//external gridcode trip (Now coming from missing phase current/ high current unbalance).
IF set.e_InverterMode = eInvertermodes.Afe OR setMaster.b_ExtgridCodeTrip THEN
	ton_GridCodeTripDelay(IN := b_extGridCodetrip);
	setMaster.b_ExtgridCodeTrip := ton_GridCodeTripDelay.Q;
	setSlave.b_ExtgridCodeTrip := ton_GridCodeTripDelay.Q;
END_IF

//calculate internal loss offset
r_ActiveLossOffset := r_APloss;
r_ReactiveLossOffset:= r_RPloss + st_params.r_ReactiveOffset;


ton_RampDisabled(IN := get.b_StartedState);
//Gross power: requested + internal loss 
r_grossActivePower := set.r_ActivePower * st_params.r_ActiveSetpointGain - r_ActiveLossOffset;
fb_ramp_Pset(IN := r_grossActivePower, SETtoIN := ton_RampDisabled.Q);
//magic reactive fix to the inverter:P
//SEL(set.r_ReactivePower < 0, -0.00039, -0.0007) * -set.r_ReactivePower + 1;
r_grossReactivePower := st_params.r_ReactiveSetpointGain * set.r_ReactivePower - r_ReactiveLossOffset;
fb_ramp_Qset(IN := r_grossReactivePower, SETtoIN := ton_RampDisabled.Q, SetZero:= NOT get.b_StartedState);


//Powerlimiting mode ugrid
PowerLimitingMode(
	enable := get.b_InverterGridFormingMode AND NOT set.b_DisableShifting,
	PowerLimitingMode := set.e_PowerLimitingMode,
	ActivePower := get.r_ActivePower,
	MaxPower := set.r_Pmax,
	MinPower := set.r_Pmin,
	ShiftHoldTimeRemaining => get.t_ShiftHoldTimeRemaining,
	Active	=> get.Events.b_PlimitShiftingActive,
	Pmax => r_PmaxFinal,
	Pmin => r_PminFinal,
	FreqOffset => r_PLMfreqOffset,
	VoltOffset => r_PLMvoltOffset,
	st_params := st_params.FreqVoltageShift,
	);
	
//Max Charge Power
SetMaster.r_Pmin := r_PminFinal * r_PM1Load;
SetSlave.r_Pmin := r_PminFinal * r_PM2Load;
//Max Discharge Power
SetMaster.r_Pmax := r_PmaxFinal * r_PM1Load;
SetSlave.r_Pmax := r_PmaxFinal * r_PM2Load;
//Max AC current limit (first reactive limits, then active);
SetMaster.r_ACcurrentLimit := set.r_ACcurrentLimit * r_PM1Load;
SetSlave.r_ACcurrentLimit:= set.r_ACcurrentLimit * r_PM2Load;

//ActivePower
setMaster.r_ActivePower := SEL(set.r_Pmax = 0 AND fb_ramp_Pset.Q > 0, fb_ramp_Pset.Q * r_PM1Load, st_params.i_ChargeOnlyIdlePower); 
setSlave.r_ActivePower := fb_ramp_Pset.Q * r_PM2Load; 


//Set Reactive Power
setMaster.r_ReactivePower := fb_ramp_Qset.Q * r_PM1Load;// fb_ramp_Qset.Q  // fb_ramp_Qset.Q * r_PM1Load;
setSlave.r_ReactivePower := fb_ramp_Qset.Q * r_PM2Load; //fb_ramp_Qset.Q * r_PM2Load;

//Overcurrent factor
setMaster.r_overcurrentFactor := CoolingDerating();
setSlave.r_overcurrentFactor := CoolingDerating();

//Max power change rate
SetMaster.i_PowerChangeRate := st_params.i_MaxPowerChangeRate; //limit to 300%/s 
SetSlave.i_PowerChangeRate := st_params.i_MaxPowerChangeRate;

//set frequency to inverter
r_FreqDeltaLOM := FreqPulseDelta(LOM.b_enable AND settings.MachineParams.Powerstack.LOM.EnablePowerPulse,
								PulseSize := st_params.LOM.PowerPulseSize,
								Droop := get.r_FrequencyDroop, 
								DetectionTime := SEL(st_params.LOM.ForceSlowDetection, st_params.LOM.DetectionTimeFast_ms, st_params.LOM.DetectionTimeSlow_ms)
								);


		
								
setMaster.r_NomFrequency := set.r_NominalOutputFrequency + r_FreqDeltaLOM + r_PLMfreqOffset;
SetSlave.r_NomFrequency := set.r_NominalOutputFrequency + r_FreqDeltaLOM + r_PLMfreqOffset;


//set voltage to inverter
setMaster.r_NomVoltage := set.r_NominalOutputVoltage + r_PLMVoltOffset;
SetSlave.r_NomVoltage := set.r_NominalOutputVoltage + r_PLMvoltOffset;
END_METHOD

METHOD CoolingDerating : REAL

VAR_INST
	percentage			: REAL;
END_VAR
//Cooling derating
IF by_CoolingPowerRequest <> 2 AND get.b_ControlEnabled THEN
	percentage := LIMIT(0, 100 - st_params.ui_DeratingLimCooling, st_params.ui_OvercurrentRating);
	get.Events.b_CoolingDerating := TRUE;
ELSE
	percentage := st_params.ui_OvercurrentRating;
	get.Events.b_CoolingDerating := FALSE;
END_IF

CoolingDerating := percentage / 100;
END_METHOD

ACTION CoolingReady_active:
IF eControl <> stand_by THEN
	by_CoolingControl := 2;
END_IF

get.e_State := eStatusPowerStack.Wait_CoolingMode2;

SFCTIP := 	((by_CoolingPowerRequest > 1 AND NOT DetectConnectionLoss(TRUE)) OR 
			(eControl = stand_by AND by_CoolingPowerRequest =1)) AND NOT SFCTip;
END_ACTION

METHOD DetectConnectionLoss : BOOL
VAR_INPUT
	CurrentState		: BOOL;
END_VAR

VAR_INST
	ftrig_Input 	: F_TRIG;
	ftrig_Output 	: F_TRIG;
END_VAR
ftrig_Output(CLK := b_OutputConnected);
ftrig_Input(CLK:= b_InputConnected);

IF NOT b_OutputConnected AND ftrig_Input.Q THEN
	DetectConnectionLoss := TRUE;
END_IF


IF NOT b_InputConnected AND ftrig_Output.Q THEN
	DetectConnectionLoss := TRUE;
END_IF

IF CurrentState THEN
	DetectConnectionLoss := NOT (b_InputConnected OR b_OutputConnected);
END_IF
END_METHOD

METHOD PRIVATE DetectGridSync : BOOL
VAR_INPUT
	b_netconFB					: BOOL;
	b_InverterGridFormingMode	: BOOL;
	b_ExtGridConnected			: BOOL;
	b_ACOK						: BOOL;
	b_IsochroneMode				: BOOL;
	b_GridCodeActiveInverter 	: BOOL;
	b_GridCodeTripInverter		: BOOL;
	t_GridLostMaxTripTime		: TIME;
	t_GridOKReleaseTime			: TIME;
END_VAR

VAR_INST
	rTrigStartCommand			: R_TRIG;
	b_inverterGridCodeOK			: BOOL;
	b_AFErequested				: BOOL;
	ton_DetectionDelay			: TON := (PT := T#50MS);
	ton_DetectionDelayNoGrid	: TON := (PT := T#50MS);
	b_ExtGridCheck				: BOOL;
	tp_ExtGridLost				: TP := (PT := T#40MS);
	fTrig_ACOK					: F_TRIG;
	ton_GridLostRelease			: TON := (PT := T#0M);
	ton_GridTripDelay			: TON ;
	DisableGCtrip				: TOF := (PT:= T#1S);
END_VAR


VAR_IN_OUT
	b_Gridtied				: BOOL;
	b_GridCodeOK			: BOOL;
	b_gridCheckActive		: BOOL;
	b_ACdetected			: BOOL;
END_VAR
PowermoduleMaster.set.b_GridCodeEnable := st_params.b_GridCodesEnabled;

// update AC detected while not connected to busbar
b_ExtGridCheck := b_ExtGridConnected AND b_InverterGridFormingMode; // OLD: get.e_InverterMode = eInvertermodes.Afe;
ton_DetectionDelay(IN := NOT b_ACOK OR (b_netconFB AND NOT get.b_InverterRunning));
tp_ExtGridLost(IN := NOT b_ExtGridConnected, PT := TO_TIME(settings.GridParams.ui_GCTripMaxTripTime));
IF ton_DetectionDelay.Q OR NOT b_netconFB OR b_ExtGridCheck OR tp_ExtGridLost.Q THEN
	b_ACdetected	:= b_ACOK;
END_IF

//conditions where gridAC is not possible.
//ton_DetectionDelayNoGrid(IN := b_netconFB AND b_InverterGridFormingMode AND get.b_StartedState); // OLD: get.e_InverterMode = eInvertermodes.Afe;
//IF ton_DetectionDelayNoGrid.Q THEN
//	b_ACdetected := FALSE;
//END_IF

//Grid OK inverter statement
b_inverterGridCodeOK := NOT b_GridCodeActiveInverter OR (NOT b_GridCodeTripInverter AND b_GridCodeActiveInverter);

//disable GC Trip
DisableGCTrip(IN:= detectConnectionLoss(TRUE));


//Manual gridlost check
b_AFERequested := set.e_InverterMode = eInvertermodes.Afe;
b_gridCheckActive := b_AFERequested OR NOT b_gridCodeOK AND NOT DisableGCTrip.Q; //or not netconfb ;
//b_gridCheckActive := set.e_InverterMode = eInvertermodes.Afe AND get.b_ControlEnabled AND NOT DisableGCTrip.Q;

LOM(r_Freq := get.r_FrequencyD7, 
	r_NomFreq := set.r_NominalOutputFrequency, 
	r_Volt:= Get.r_ACVoltageD7,
	b_enable := Get.b_StartedState AND get.e_PowerMode = ePowermodes.Isochronous AND get.e_InverterMode <> eInvertermodes.Afe,
	SlowDetection:= set.b_slowLom, //only activate fast when external grid is coupled.
	st_params := st_params.LOM);

IF LOM.Q THEN
	b_gridCheckActive := TRUE;
END_IF

IF b_ACOK AND b_gridCodeOK THEN
	LOM.Reset();
END_IF


ton_GridTripDelay(IN:= NOT b_ACOK AND b_gridCheckActive, PT := t_GridLostMaxTripTime);
IF ton_GridTripDelay.Q OR NOT b_inverterGridCodeOK OR LOM.Q THEN
	b_ACdetected := FALSE;
	b_gridCodeOK := FALSE;
END_IF

get.t_GridCodeReconnectTime := ton_GridLostRelease.PT - ton_GridLostRelease.ET;

ton_GridLostRelease(
	IN := b_ACOK AND b_inverterGridCodeOK AND NOT LOM.Q AND NOT b_gridCodeOK,
	PT := SEL(b_gridCheckActive AND b_AFERequested, T#1S, t_GridOKReleaseTime)
	);

rTrigStartCommand(CLK:= eControl = start);
IF ton_GridLostRelease.Q OR NOT get.b_ControlEnabled OR DisableGCTrip.Q OR rTrigStartCommand.Q THEN
	b_gridCodeOK := TRUE;
END_IF

get.Events.b_GridCodeWarning := NOT b_gridCodeOK;
b_Gridtied := b_netconFB AND b_gridCodeOK AND b_gridCheckActive;
END_METHOD

METHOD PUBLIC EMstop : BOOL
EMstop := 
	SFCCurrentStep = 'Init' AND Netcontactor.Open() AND ShutdownFull(TRUE);
//Set internal control mode to shutdown
eControl := Shutdown;



//force SFC to init with execution of init step
SFCReset := TRUE;

IF EMstop THEN
	get.e_State := eStatusPowerStack.off;
END_IF
END_METHOD

METHOD FreqCheckPLimitUgrid : BOOL
VAR_INPUT
	b_enable			: BOOL;
	r_Frequency			: REAL;
	r_LowFreqLim		: REAL;
	r_HighFreqLim		: REAL;
	t_TriggerDelay		: TIME := T#1000MS;
END_VAR

VAR_OUTPUT
	b_LowFreqTrip		: BOOL;
	b_HighFreqTrip		: BOOL;
END_VAR

VAR_INST
	ton_TriggerDelay	: TON;
	Activate			: BOOL;
END_VAR
(*
-------INFO---------
This function is added to raise a normal shutdown before the inverter does at under/over frequency in ugrid.
this under/over frequency check is raised when the pmax or pmin limit is reached in ugrid mode resulting in frequency shift done by inverter.
To avoid a trip by inverter underfrequency, resulting in ac outage, we detect the event slightly earlier.
This creates a normal shutdown command in the error program and will keep possibility of correctly stopping the cooling supply.
If this script was not here, the under frequency trip of the inverter would be seen, leading to AC outage and this
interrupts all internal AC devices. Especially for the heatpump, this is undesirable. 
*)


activate := b_enable AND LIMIT(get.r_Pmin, get.r_ActivePower, get.r_Pmax) <> get.r_ActivePower; 
ton_triggerDelay(IN := (r_Frequency < r_LowFreqLim OR r_Frequency > r_HighFreqLim) AND activate, PT := t_TriggerDelay);

IF ton_triggerDelay.Q THEN
	b_LowFreqTrip := r_Frequency < r_LowFreqLim;
	b_HighFreqTrip := r_Frequency > r_HighFreqLim;
END_IF
END_METHOD

METHOD FreqPulseDelta : REAL
VAR_INPUT
	Enable			: BOOL;
	PulseSize		: REAL; // % of ratedpower
	Droop			: REAL;
	DetectionTime	: UINT;
END_VAR

VAR_INST
	DetectionTimeFactor	: UINT := 3; 
	FreqShift			: REAL;
	ton_PulseTime		: TON;
	b_toggleState		: BOOL;
END_VAR
(*-------INFO---------
This function is for intentionally disturbing the frequency setpoint of the inverter in a microgrid. It has been with grid and genset connected.
Testing must be done for multiple batteries in ugrid mode. The small disturbances are made on the frequency. The pulsesize is in % of rated power.
The change of the frequency therefore is relative to the droop settings and the nominal frequency setting.
The detection time and a multiplication factor gives the sweet spot of the pulse time and detection mechanism in the LOM detection.

If this puls is disabled in ugrid, the LOM detection might not function properly and
frequency might drift away in case of grid loss before transition to island mode is made.
*)

ton_PulseTime(IN := NOT ton_pulseTime.Q, PT := TO_TIME(detectionTime*DetectionTimeFactor)); //must be bigger than detection time. factor 5 seems fine.

IF ton_pulseTime.Q THEN
	b_ToggleState := NOT b_toggleState;
END_IF


FreqShift := PulseSize / 100 * settings.GridParams.r_GridNominalFrequency * Droop / 100; 
IF enable THEN
	FreqPulseDelta := SEL(b_toggleState, -1, 1) * FreqShift;
ELSE
	FreqPulseDelta := 0;
END_IF
END_METHOD

METHOD PUBLIC GetDiagnostics
VAR_IN_OUT
	AddError		: ARRAY [*] OF FB_AddErrorST;
	a_ActiveEvents	: ARRAY [*] OF ST_ErrorStruct;
	w_Index			: WORD;
END_VAR

VAR_INST
	varString		: STRING;
END_VAR
(*POWERSTACK*)
	//Warnings
	(*DC voltage diff*) 	AddError[w_Index](
			b_ErrorTrig			:= Get.Events.b_DCdeviationHigh,
			out_ST_Error			:= a_ActiveEvents[w_Index],
			w_ErrorID					:= 1,
			e_ObjectID				:= eObject_ID.PowerStack,
			s_Message				:= 'DC voltage difference between powermodules high',
			e_sev					:= eseverity.Warning
			);
		w_Index := w_Index +1;
	
	(*Temperature*) 			AddError[w_Index](
			b_ErrorTrig			:= Get.Events.b_TemperatureDeviationHigh,
			out_ST_Error			:= a_ActiveEvents[w_Index],
			w_ErrorID					:= 2,
			e_ObjectID				:= eObject_ID.PowerStack,
			s_Message				:= 'temperature difference between powermodules high',
			e_sev					:= eseverity.Warning,
			b_AutoClear			:= TRUE,
		);
		w_Index := w_Index +1;
		
	(*UnderFreq limit exceeded*)	AddError[w_Index](
			b_ErrorTrig				:= Get.Events.b_UnderFreqFault ,
			out_ST_Error			:= a_ActiveEvents[w_Index],
			w_ErrorID				:= 3,
			e_ObjectID				:= eObject_ID.PowerStack,
			s_Message				:= 'under frequency trip',
			e_sev					:= eseverity.normalshutdown
		);
		w_Index := w_Index +1;	
		
	(*OverFreq limit exceeded*)		AddError[w_Index](
			b_ErrorTrig				:= Get.Events.b_OverFreqFault,
			out_ST_Error			:= a_ActiveEvents[w_Index],
			w_ErrorID				:= 4,
			e_ObjectID				:= eObject_ID.PowerStack,
			s_Message				:= 'over frequency trip',
			e_sev					:= eseverity.normalshutdown
		);
		w_Index := w_Index +1;	
		
	(*Cooling derating*)	AddError[w_Index](
			b_ErrorTrig			:=  get.Events.b_CoolingDerating,
			out_ST_Error			:= a_ActiveEvents[w_Index],
			w_ErrorID				:= 5,
			s_Message				:= 'Cooling system derating causing inverter output to be limited',
			e_sev					:= eseverity.warning,
			b_autoclear				:= TRUE,
		);
		w_Index := w_Index +1;

	(*SFC Timeout*)	AddError[w_Index](
			b_ErrorTrig				:= SFCerror,
			out_ST_Error			:= a_ActiveEvents[w_Index],
			w_ErrorID				:= 6,
			e_ObjectID				:= eObject_ID.PowerStack,
			s_Message				:= CONCAT('SFC error at step: ', s_errorstep),
			e_sev					:= eseverity.NormalShutdown
		);
		w_Index := w_Index +1;
		
		
(*Start inhibit*)	AddError[w_Index](
			b_ErrorTrig				:= NOT get.b_StartEnabled AND set.e_InverterMode = eInvertermodes.Afe,
			out_ST_Error			:= a_ActiveEvents[w_Index],
			w_ErrorID				:= 8,
			s_Message				:= CONCAT('Inverter starting in grid following mode inhibited, ',SEL(NOT get.b_GridCodeOK AND get.b_GridCodeCheckActive, 'waiting for grid AC','waiting for gridcode release')),
			e_sev					:= eseverity.info,
			b_autoclear				:= TRUE,
		);
		w_Index := w_Index +1;
		
(*Start inhibit*)	AddError[w_Index](
			b_ErrorTrig			:= NOT get.b_StartEnabled AND set.e_InverterMode = eInvertermodes.Island,
			out_ST_Error			:= a_ActiveEvents[w_Index],
			w_ErrorID				:= 9,
			s_Message				:= 'Inverter starting in grid forming mode inhibited, disconnect AC from busbar',
			e_sev					:= eseverity.info,
			b_autoclear				:= TRUE,
		);
		w_Index := w_Index +1;
		
	(*Overvoltage fault*)	AddError[w_Index](
			b_ErrorTrig			:= get.Events.b_OverVoltageFault,
			out_ST_Error			:= a_ActiveEvents[w_Index],
			w_ErrorID				:= 10,
			s_Message				:= 'Overvoltage fault', //10-12-2024: change to normalshutdown once verified
			e_sev					:= eseverity.warning,
			b_autoclear				:= FALSE,
		);
		w_Index := w_Index +1;
		
	(*underVoltage fault*)	AddError[w_Index](
			b_ErrorTrig			:= get.Events.b_underVoltageFault,
			out_ST_Error			:= a_ActiveEvents[w_Index],
			w_ErrorID				:= 11,
			s_Message				:= 'Undervoltage fault',
			e_sev					:= eseverity.warning, // 10-12-2024: change to normalshutdown once verified 
			b_autoclear				:= FALSE,
		);
		w_Index := w_Index +1;
		
	(*Overvoltage warning*)	AddError[w_Index](
			b_ErrorTrig			:= get.Events.b_OverVoltageFault,
			out_ST_Error			:= a_ActiveEvents[w_Index],
			w_ErrorID				:= 12,
			s_Message				:= 'Overvoltage warning',
			e_sev					:= eseverity.warning,
			b_autoclear				:= TRUE,
		);
		w_Index := w_Index +1;
		
	(*underVoltage fault*)	AddError[w_Index](
			b_ErrorTrig			:= get.Events.b_underVoltageFault,
			out_ST_Error			:= a_ActiveEvents[w_Index],
			w_ErrorID				:= 13,
			s_Message				:= 'Undervoltage warning',
			e_sev					:= eseverity.warning,
			b_autoclear				:= TRUE,
		);
		w_Index := w_Index +1;

		(*Overvoltage warning*)	AddError[w_Index](
			b_ErrorTrig			:= get.Events.b_TemperatureFault,
			out_ST_Error			:= a_ActiveEvents[w_Index],
			w_ErrorID				:= 14,
			s_Message				:= 'Temperature fault',
			e_sev					:= eseverity.warning,
			b_autoclear				:= TRUE,
		);
		w_Index := w_Index +1;
		
	(*underVoltage fault*)	AddError[w_Index](
			b_ErrorTrig			:= get.Events.b_TemperatureWarning,
			out_ST_Error			:= a_ActiveEvents[w_Index],
			w_ErrorID				:= 15,
			s_Message				:= 'Temperature warning',
			e_sev					:= eseverity.warning,
			b_autoclear				:= TRUE,
		);
		w_Index := w_Index +1;
		
(*Plimit warning*)	AddError[w_Index](
			b_ErrorTrig				:= get.Events.b_PlimitShutdownWarning,
			out_ST_Error			:= a_ActiveEvents[w_Index],
			w_ErrorID				:= 16,
			s_Message				:= CONCAT(CONCAT('Power limit reached, shutdown in ', TO_STRING(get.Events.ui_shutdownRemainingTime)),'s'),
			e_sev					:= eseverity.warning,
			b_autoclear				:= TRUE,
		);
		w_Index := w_Index +1;
		
(*Plimit shutdown*)	AddError[w_Index](
			b_ErrorTrig				:= get.Events.b_PlimitShutdown,
			out_ST_Error			:= a_ActiveEvents[w_Index],
			w_ErrorID				:= 17,
			s_Message				:= 'Power limit shutdown',
			e_sev					:= eseverity.normalshutdown,
			b_autoclear				:= TRUE,
		);
		w_Index := w_Index +1;
		
(*Plimit shifting *)	AddError[w_Index](
			b_ErrorTrig				:= get.Events.b_PlimitShiftingActive,
			out_ST_Error			:= a_ActiveEvents[w_Index],
			w_ErrorID				:= 18,
			s_Message				:= CONCAT(CONCAT(TO_STRING(set.e_PowerLimitingMode), ' active, output on hold for: '), TO_STRING(get.t_ShiftHoldTimeRemaining)),
			e_sev					:= eseverity.Warning,
			b_autoclear				:= TRUE,
		);
		w_Index := w_Index +1;

		
IF get.b_GridACdetected THEN
	varstring := CONCAT('gridcode disconnect active, reconnecting in: ', TO_STRING(get.t_GridCodeReconnectTime));
ELSE
	varstring := 'gridcode disconnect active, reset to reconnect in island mode';
END_IF
		
(*Gridcode disconnect *)	AddError[w_Index](
			b_ErrorTrig				:= get.Events.b_GridCodeWarning,
			out_ST_Error			:= a_ActiveEvents[w_Index],
			w_ErrorID				:= 19,
			s_Message				:= varstring,
			e_sev					:= eseverity.warning,
			b_autoclear				:= TRUE,
		);
		w_Index := w_Index +1;



(*INSERT NESTED OBJECTS*)
Netcontactor.GetDiagnostics(AddError := AddError, a_activeEvents:= a_ActiveEvents, w_Index:= w_Index);
PowermoduleMaster.GetDiagnostics(AddError := AddError, a_activeEvents:= a_ActiveEvents, w_Index:= w_Index);
PowermoduleSlave.GetDiagnostics(AddError := AddError, a_activeEvents:= a_ActiveEvents, w_Index:= w_Index);
END_METHOD

METHOD GetWearCounters : BOOL
VAR_INST
	RightNetContactor	:	FB_Varlogger;
	LeftNetContactor	:	FB_Varlogger;
	
	MasterPmMCCB		:	FB_Varlogger;
	MasterPmDCMain		:	FB_Varlogger;
	MasterPmPrecharge	:	FB_Varlogger;
	MasterPMACFanHrs	:	FB_Varlogger;		
	
	SlavePmMCCB			:	FB_Varlogger;
	SlavePmDCMain		:	FB_Varlogger;
	SlavePmPrecharge	:	FB_Varlogger;
	SlavePMACFan		:	FB_Varlogger;
	
	SlowDataTimer				:	TON := (PT := T#30M);
	
	initdone		:	Bool;
END_VAR
SlowDataTimer(in := NOT SlowDataTimer.Q);

IF get.PowermoduleMaster.w_OperationHours > 0 THEN
	Wearlogging.SetInteger(eLogItemGroupID.PowerStack, 	'MstrInvHrs', 				eLogTypes.WriteValue, 		WORD_TO_LINT(get.PowermoduleMaster.w_OperationHours));
END_IF
Wearlogging.SetFloat(eLogItemGroupID.PowerStack, 	'MstrMaxDischCurrentEver', 	eLogTypes.KeepHighestValue, REAL_TO_LREAL(get.PowermoduleMaster.r_ACCurrent));
Wearlogging.SetFloat(eLogItemGroupID.PowerStack, 	'MstrMaxChargeCurrentEver', eLogTypes.KeepLowestValue, 	REAL_TO_LREAL(get.PowermoduleMaster.r_AcCurrent));
		
												
MasterPmMCCB(			TriggerInput := get.PowermoduleMaster.b_MccbFb, 
						LogItemGroup :=  eLogItemGroupID.PowerStack, 
						LogItemName := 'MstrMCCBCnt', 
						LogType := eLogTypes.TrackCycles);	
						
MasterPmDCMain(			TriggerInput := get.PowermoduleMaster.b_DCcontactorFb, 
						LogItemGroup :=  eLogItemGroupID.PowerStack, 
						LogItemName := 'MstrDcMainCnt', 
						LogType := eLogTypes.TrackCycles);							

MasterPmPrecharge(		TriggerInput := get.PowermoduleMaster.b_PrechargeContactor, 
						LogItemGroup :=  eLogItemGroupID.PowerStack, 
						LogItemName := 'MstrDcPrechargeCnt', 
						LogType := eLogTypes.TrackCycles);		

MasterPMACFanHrs(		TriggerInput := get.PowermoduleMaster.b_FanFb, 
						LogItemGroup :=  eLogItemGroupID.PowerStack, 
						LogItemName := 'MstrAcFanHrs', 
						LogType := eLogtypes.TrackOnTime);	



					
IF b_doublePowermodule THEN
	Wearlogging.SetInteger(eLogItemGroupID.PowerStack, 	'SlvInvHrs', 				eLogTypes.WriteValue, 		WORD_TO_LINT(get.PowermoduleSlave.w_OperationHours));
	Wearlogging.SetFloat(eLogItemGroupID.PowerStack, 	'SlvMaxDischCurrentEver', 	eLogTypes.KeepHighestValue, REAL_TO_LREAL(get.PowermoduleSlave.r_ACCurrent));
	Wearlogging.SetFloat(eLogItemGroupID.PowerStack, 	'SlvMaxChargeCurrentEver', 	eLogTypes.KeepLowestValue, 	REAL_TO_LREAL(get.PowermoduleSlave.r_AcCurrent));		
												
	SlavePmMCCB(			TriggerInput := get.PowermoduleSlave.b_MccbFb, 
							LogItemGroup :=  eLogItemGroupID.PowerStack, 
							LogItemName := 'SlvMCCBCnt', 
							LogType := eLogTypes.TrackCycles);	
							
	SlavePmDCMain(			TriggerInput := get.PowermoduleSlave.b_DCcontactorFb, 
							LogItemGroup :=  eLogItemGroupID.PowerStack, 
							LogItemName := 'SlvDcMainCnt', 
							LogType := eLogTypes.TrackCycles);							
	
	SlavePmPrecharge(		TriggerInput := get.PowermoduleSlave.b_PrechargeContactor, 
							LogItemGroup :=  eLogItemGroupID.PowerStack, 
							LogItemName := 'SlvDcPrechargeCnt', 
							LogType := eLogTypes.TrackCycles);		
	
	SlavePMACFan(			TriggerInput := get.PowermoduleSlave.b_FanFb, 
							LogItemGroup :=  eLogItemGroupID.PowerStack, 
							LogItemName := 'SlvAcFanHrs', 
							LogType := eLogTypes.TrackOnTime);	
END_IF


RightNetContactor(		TriggerInput := get.Netcontactor.b_NetcontRightFb, 
						LogItemGroup :=  eLogItemGroupID.PowerStack, 
						LogItemName := 'NetcRightCnt', 
						LogType := eLogTypes.TrackCycles);		
												
LeftNetContactor(		TriggerInput := get.Netcontactor.b_NetcontLeftFb, 
						LogItemGroup :=  eLogItemGroupID.PowerStack, 
						LogItemName := 'NetcLeft', 
						LogType := eLogTypes.TrackCycles);	
						
IF NOT initdone THEN
	Wearlogging.SetFloat(eLogItemGroupID.General, 	'nameplatePowerCapacity', 	eLogTypes.WriteValue, 	TO_DINT(SEL(settings.Configuration.b_DoublePowerModule, 360, 720)));
	initdone := TRUE;		
END_IF
END_METHOD

METHOD PRIVATE InternalAcCheck : BOOL
VAR_INPUT
	r_ACVoltage	: REAL;
	r_ACFreq	: REAL;
END_VAR

VAR_INST
	b_VoltageOK				: BOOL;
	b_FrequencyOK			: BOOL;
	tof_ReleaseACNOK		: TOF := (PT:= T#2S);
	
	tof_MaxRetryTimeOut		: Tof := (PT:= T#60S);
	ton_ResetRetries		: TON := (PT:= T#60S);
	by_maxRetries			: BYTE := 5;
	by_retries				: BYTE;
	r_trigOK				: r_TRIG;
END_VAR
b_VoltageOK	:= LIMIT(350, r_ACVoltage, 450) = r_ACVoltage;
b_FrequencyOK :=  LIMIT(45, r_ACFreq, 65) = r_ACFreq;

tof_ReleaseACNOK(IN:= b_VoltageOK AND b_FrequencyOK); 
	
r_trigOK(CLK := tof_ReleaseACNOK.Q);
IF r_trigOK.Q THEN
	by_Retries := by_retries + 1;
END_IF
IF by_Retries > by_MaxRetries THEN
	by_Retries := 0;
	tof_MaxRetryTimeOut(IN := TRUE);
ELSE
	tof_MaxRetryTimeOut(IN := FALSE);
END_IF
	
InternalAcCheck := tof_ReleaseACNOK.Q AND NOT tof_MaxRetryTimeOut.Q;
ton_ResetRetries(IN:= InternalAcCheck);
IF ton_ResetRetries.Q THEN
	by_Retries := 0;
END_IF
END_METHOD

METHOD PowerLimitingMode;
VAR_INPUT
	enable					: BOOL;
	PowerLimitingMode		: ePLM;
	ActivePower				: REAL;
	MaxPower				: REAL;
	MinPower				: REAL;
END_VAR
VAR_IN_OUT CONSTANT
	st_params : ST_powerstack_ShiftingParams;
END_VAR

VAR_INST
	tof_shiftHoldTime	: Tof := (PT := T#20M);
	tPulseRate			: TIME := T#100MS;
	tonIncreasePulse	: TON := (PT := T#100MS);
	OffsetCounter		: CTUD;
	i_counterValue		: INT;
	PDeadband			: REAL := 3;
	PmaxReached			: BOOL;
	PminReached			: BOOL;
	Nolimit				: BOOL;
	
	MaxVoltOffsetUp		: REAL := 40;
	MaxVoltOffsetDown	: REAL := 40;
	
	MaxFreqOffsetUp		: REAL := 2.5;
	MaxFreqOffsetDown	: REAL := 2.5;
	
	r_FreqStepUp	: REAL := 0.1; // hz/s
	r_FreqStepDown	: REAL := 0.1; // hz/s
	r_FreqStepActual: REAL ;
	r_VoltStepUp	: REAL := 0.1; // V/s
	r_VoltStepDown 	: REAL := 0.1;
	r_VoltStepActual: REAL ;
	
	w_CounterSteps		: WORD := 1000;
	ton_InitialPmaxDelay	: TON := (PT := T#1S);
	ton_InitialPminDelay	: TON := (PT := T#1S);
	ton_shutdownTimer	: TON := (PT := T#1M);
	shutdownTrigger		: BOOL;
END_VAR

VAR_OUTPUT
	ShiftHoldTimeRemaining 	: TIME;
	Active				: BOOL;
	Pmax				: REAL;
	Pmin				: REAL;
	FreqOffset			: REAL;
	VoltOffset			: REAL;
END_VAR
IF NOT enable THEN
	Pmax := MaxPower;
	Pmin := MinPower;
	get.Events.b_PlimitShutdownWarning := FALSE;
	get.Events.b_PlimitShutdown := FALSE;
	active := FALSE;
	ShiftHoldTimeRemaining := st_params.ShiftingHoldTime;
	RETURN;
END_IF

shutdownTrigger	:= FALSE;
ton_InitialPmaxDelay(in := ActivePower > MAX(MaxPower, PDeadband), pt := st_params.InitialOverloadDelay);
ton_InitialPminDelay(in := ActivePower < MIN(MinPower, -PDeadband), pt := st_params.InitialOverloadDelay);

PmaxReached := ton_InitialPmaxDelay.Q;
PminReached	:= ton_InitialPminDelay.Q;

Nolimit := NOT PmaxReached AND NOT PminReached;

//max voltage offsets based on grid settings
MaxVoltOffsetUp := LIMIT(settings.GridParams.r_GridNominalVoltage, st_params.VoltMaxPu * settings.GridParams.r_GridNominalVoltage, settings.GridParams.r_GridvoltageMax) - settings.GridParams.r_GridNominalVoltage;
MaxVoltOffsetDown := settings.GridParams.r_GridNominalVoltage - LIMIT(settings.GridParams.r_GridvoltageMin, st_params.VoltMinPu * settings.GridParams.r_GridNominalVoltage, settings.GridParams.r_GridNominalVoltage);
r_VoltStepUp := MaxVoltOffsetUp / MAX(1, w_CounterSteps);
r_VoltStepDown := MaxVoltOffsetDown/ MAX(1, w_CounterSteps);
r_VoltStepActual := SEL(i_countervalue < 0, r_VoltStepUp, r_VoltStepDown);

//max frequency offsets based on grid settings
MaxFreqOffsetUp := LIMIT(settings.GridParams.r_GridNominalFrequency, st_params.FreqMaxPu * settings.GridParams.r_GridNominalFrequency, settings.GridParams.r_GridFrequencyMax) - settings.GridParams.r_GridNominalFrequency;
MaxFreqOffsetDown := settings.GridParams.r_GridNominalFrequency - LIMIT(settings.GridParams.r_GridFrequencyMin, st_params.FreqMinPu * settings.GridParams.r_GridNominalFrequency, settings.GridParams.r_GridNominalFrequency);
r_FreqStepUp := MaxFreqOffsetUp / MAX(1, w_CounterSteps);
r_FreqStepDown := MaxFreqOffsetDown / MAX(1, w_CounterSteps);
r_FreqStepActual := SEL(i_countervalue < 0, r_FreqStepUp, r_FreqStepDown);

//If shifting is done and limit is released. Hold current counter for 20 min, before reducing.
tof_shiftHoldTime(IN := (i_countervalue <> 0 AND NOT Nolimit), PT := st_params.ShiftingHoldTime);

//pulse Timer
tonIncreasePulse(IN := NOT tonIncreasePulse.Q, PT := tPulseRate);

OffsetCounter(
	CU := ((PminReached OR (i_countervalue < 0 AND Nolimit AND NOT tof_shiftHoldTime.Q)) AND tonIncreasePulse.Q) AND NOT OffsetCounter.QU,
	CD := ((PmaxReached OR (i_countervalue > 0 AND Nolimit AND NOT tof_shiftHoldTime.Q)) AND tonIncreasePulse.Q) AND NOT OffsetCounter.QD,
	LOAD := NOT get.b_StartedState,
	PV := SEL(get.b_StartedState, w_CounterSteps, w_CounterSteps*2));
i_countervalue := OffsetCounter.CV - w_CounterSteps;

CASE PowerLimitingMode OF
	ePLM.FreqShift: //default controlled by inverters
		Pmax := get.r_RatedPower;
		Pmin := -get.r_RatedPower;
		FreqOffset := LIMIT(-MaxFreqOffsetDown, r_FreqStepActual * i_countervalue, MaxFreqOffsetUp);
		
	ePLM.VoltShift:
		VoltOffset := LIMIT(-MaxVoltOffsetDown, r_VoltStepActual * i_countervalue, MaxVoltOffsetUp);
		Pmax := get.r_RatedPower;
		Pmin := -get.r_RatedPower;
		
	ePLM.FreqVoltShift:
		VoltOffset := LIMIT(-MaxVoltOffsetDown, r_VoltStepActual * i_countervalue, MaxVoltOffsetUp);
		FreqOffset := LIMIT(-MaxFreqOffsetDown, r_FreqStepActual * i_countervalue, MaxFreqOffsetUp);
		Pmax := get.r_RatedPower;
		Pmin := -get.r_RatedPower;
		
	ePLM.Shutdown:
		shutdownTrigger	:= NOT Nolimit;
		Pmax := get.r_RatedPower;
		Pmin := -get.r_RatedPower;	
END_CASE

ton_shutdownTimer(IN:= shutdownTrigger AND get.b_StartedState, PT := st_params.ShutdownDelay);
IF get.Events.b_PlimitShutdownWarning THEN
	get.Events.ui_shutdownRemainingTime := TO_UINT(TO_REAL(ton_shutdownTimer.PT - ton_shutdownTimer.ET)/ 1000);
END_IF

//outputs and events
Active := i_countervalue <> 0 AND PowerLimitingMode <> ePLM.Shutdown;
ShiftHoldTimeRemaining := tof_shiftHoldTime.PT - tof_shiftHoldTime.ET;
get.Events.b_PlimitShutdownWarning := ton_shutdownTimer.IN;
get.Events.b_PlimitShutdown := ton_shutdownTimer.Q;
END_METHOD

METHOD PUBLIC Reset : BOOL
Reset := Netcontactor.Reset() AND PowermoduleMaster.Reset() AND PowerModuleSlave.Reset() AND get.e_State <> eStatusPowerstack.fault;

standbyDeactivateState := FALSE;
get.b_GridCodeOK := TRUE;
//rs_Stop.RESET1 := TRUE;
//rs_StartUp.RESET1:= TRUE;	
//rs_Shutdown.RESET1:= TRUE;
END_METHOD

METHOD PRIVATE SetEvents
VAR_IN_OUT
	events							: ST_PowerStack_Events;
END_VAR

VAR_IN_OUT CONSTANT
	st_params						: ST_Powerstack_Params;
END_VAR


VAR
	r_DCVoltageDeviation			: REAL := 0.02; //2%
	r_TemperatureDeviation			: REAL:= 10; // 10C
END_VAR

VAR_INST
	tp_ACdetectionCheck				: TON:= (PT:=T#2S);
END_VAR
IF b_doublePowermodule THEN
	//DC Voltage Deviation higher than 2% between powermodules
	events.b_DCdeviationHigh:= ABS(get.PowermoduleMaster.r_DCVoltage - get.PowermoduleSlave.r_DCVoltage) > get.r_DCVoltage * r_DcVoltageDeviation;
	
	//Temperature Deviation between highest temperature in powermodules higher than 10C
	events.b_temperatureDeviationHigh:= ABS(get.PowermoduleMaster.r_TemperatureMax - get.PowermoduleSlave.r_TemperatureMax) > r_TemperatureDeviation;
	
	//slave warning and faults
	events.b_SlaveFault := get.PowermoduleSlave.Events.b_GeneralFaultFlag;
	events.b_SlaveWarning := get.PowermoduleSlave.Events.b_GeneralWarningFlag;

END_IF

//Master warning and faults
events.b_MasterFault := get.PowermoduleMaster.Events.b_GeneralFaultFlag;
events.b_MasterWarning := get.PowermoduleMaster.Events.b_GeneralWarningFlag;
events.b_OvercurrentFault := get.PowermoduleMaster.Events.b_F1OverCurrent OR get.PowermoduleSlave.Events.b_F1OverCurrent;
events.b_OvercurrentWarning := get.r_LoadPercent > get.r_OvercurrentValueAct * 100;
events.b_OvervoltageFault :=  get.PowermoduleMaster.Events.b_F2OverVoltage OR get.PowermoduleSlave.Events.b_F2OverVoltage;
events.b_OvervoltageWarning := get.r_ACVoltageD7 > settings.GridParams.r_GridvoltageMax;
events.b_TemperatureFault := PowermoduleMaster.GetTemperatureEvents(FALSE) OR
	PowermoduleSlave.GetTemperatureEvents(FALSE);
events.b_TemperatureWarning := PowermoduleMaster.GetTemperatureEvents(TRUE) OR
	PowermoduleSlave.GetTemperatureEvents(TRUE);
events.b_startupTimeOut := SFCerror;

FreqCheckPLimitUgrid(
	b_enable := get.b_StartedState AND get.e_InverterMode <> eInvertermodes.Afe AND get.e_PowerMode <> ePowermodes.Isochronous, 
	r_Frequency := get.r_FrequencySupply,
	r_LowFreqLim := st_params.r_FreqLowLimit,
	r_HighFreqLim := st_params.r_FreqHighLimit,
	t_TriggerDelay := TO_TIME(st_params.ui_FreqLimitTripDelay),
	b_LowFreqTrip => events.b_UnderFreqFault,
	b_HighFreqTrip => events.b_OverFreqFault);
END_METHOD

METHOD Shutdowncmd : BOOL
eControl := Shutdown;
//if SFC transition occurs, give feedback.
SFCreset := TRUE;
Shutdowncmd := FALSE;

get.e_State := eStatusPowerStack.shutdown; 
by_CoolingControl := 0;

IF b_InternalACRequired THEN
	get.e_State := eStatusPowerStack.Cooling_Shutdown;
	standbyDeactivateState := TRUE;
		powermodulemaster.Run(Powermode := ePowermodes.Isochronous, InverterMode := eInvertermodes.Microgrid, TRUE );
		IF netcontactor.Open() THEN;
			powermodulemaster.Run(Powermode := ePowermodes.DroopZeroStart, InverterMode := eInvertermodes.Microgrid, TRUE);
			Shutdowncmd	:= TRUE;
		END_IF
	//END_IF
ELSE
	IF ShutdownFull(FALSE)  THEN;
		IF Netcontactor.Open() THEN
			Shutdowncmd	:= TRUE;
			get.e_State := eStatusPowerStack.off;
		END_IF
	END_IF
	
END_IF
	
//	CASE by_CoolingPowerRequest OF // when cooling system allows, all power is killed
//		0: //off
//			by_CoolingControl := 0;
//				IF ShutdownFull(FALSE)  THEN ;
//					IF NOT st_params.b_StandbyEnable THEN
//						IF Netcontactor.Open() THEN
//							Shutdowncmd	:= TRUE;
//							get.e_State := eStatusPowerStack.off;
//						END_IF
//					ELSE			
//						IF NOT get.b_ACDetected THEN
//							Netcontactor.Open();
//						END_IF
//						Shutdowncmd	:= TRUE;
//						get.e_State := eStatusPowerStack.off;
//					END_IF
//				END_IF	
		
//		1, 2: //limited 	
////			IF false then //get.b_GridACdetected THEN //get.b_ACDetected THEN 
////				by_CoolingControl := 0;
////				Shutdowncmd := ShutdownFull(FALSE);
////			ELSE
//				by_CoolingControl := 1;
//				PowerModuleSlave.Shutdown(b_force := FALSE);
//				Shutdowncmd := Netcontactor.Open();
//			//END_IF// if cooling system still wants power AND AC grid is available	
//	END_CASE				

//Shutdowncmd := get.e_Status = eStatusPowerStack.off OR get.e_Status = eStatusPowerStack.init;
END_METHOD

METHOD PRIVATE ShutdownFull : BOOL
VAR_INPUT
	b_force : BOOL;
END_VAR

VAR_INST
	shutdownfb: BOOL;
	ton_ShutdownTimeOut				: TON:= (PT:=T#30S);
END_VAR
shutdownfb := PowermoduleMaster.Shutdown(b_force) AND PowermoduleSlave.Shutdown(b_force);
IF shutdownfb THEN
	st_InternalPsuSupplyRequest.b_Demand_HVDC := FALSE;
	st_InternalPsuSupplyRequest.b_Demand_24V := FALSE;
END_IF

ton_ShutdownTimeOut(IN := NOT shutdownfb, Q => get.Events.b_ShutdownTimeOut);


ShutdownFull := shutdownfb;
END_METHOD

METHOD Standbycmd : BOOL
VAR_INPUT
END_VAR
IF NOT(get.e_State = eStatusPowerstack.fault) THEN
	eControl := stand_by;
END_IF

//if SFC transition occurs, give feedback.
Standbycmd := get.e_State = eStatusPowerstack.Standby_GridSupply OR get.e_State = eStatusPowerstack.Standby_GridSupply;
END_METHOD

METHOD PUBLIC Startcmd : BOOL
IF get.b_StartEnabled THEN
	eControl := start;
END_IF

//if we get to status running, give feedback.
Startcmd := get.e_State = eStatusPowerStack.running OR get.e_State = eStatusPowerStack.idle;
END_METHOD

METHOD StartingEnable : BOOL
VAR_INPUT
END_VAR
VAR_INST
	b_startcondAFE : BOOL;
	b_startcondUgrid: BOOL;
	b_startcondNoFaults: BOOL;
	b_startcondIsland: BOOL;
END_VAR
b_StartcondAFE := set.e_InverterMode = eInvertermodes.Afe AND get.b_GridACdetected;
b_startcondUgrid:= set.e_InverterMode = eInvertermodes.microgrid;

b_startcondNoFaults := NOT(get.e_State = eStatusPowerstack.fault OR powermodulemaster.get.Events.b_GeneralFaultFlag OR powermoduleslave.get.Events.b_GeneralFaultFlag);
b_startcondIsland:=  set.e_InverterMode = eInvertermodes.Island AND NOT get.b_GridACdetected;

StartingEnable := (b_StartcondAFE OR b_startcondUgrid OR b_startcondIsland) AND b_startcondNoFaults OR get.b_StartedState;
END_METHOD

ACTION StartStopSFC:
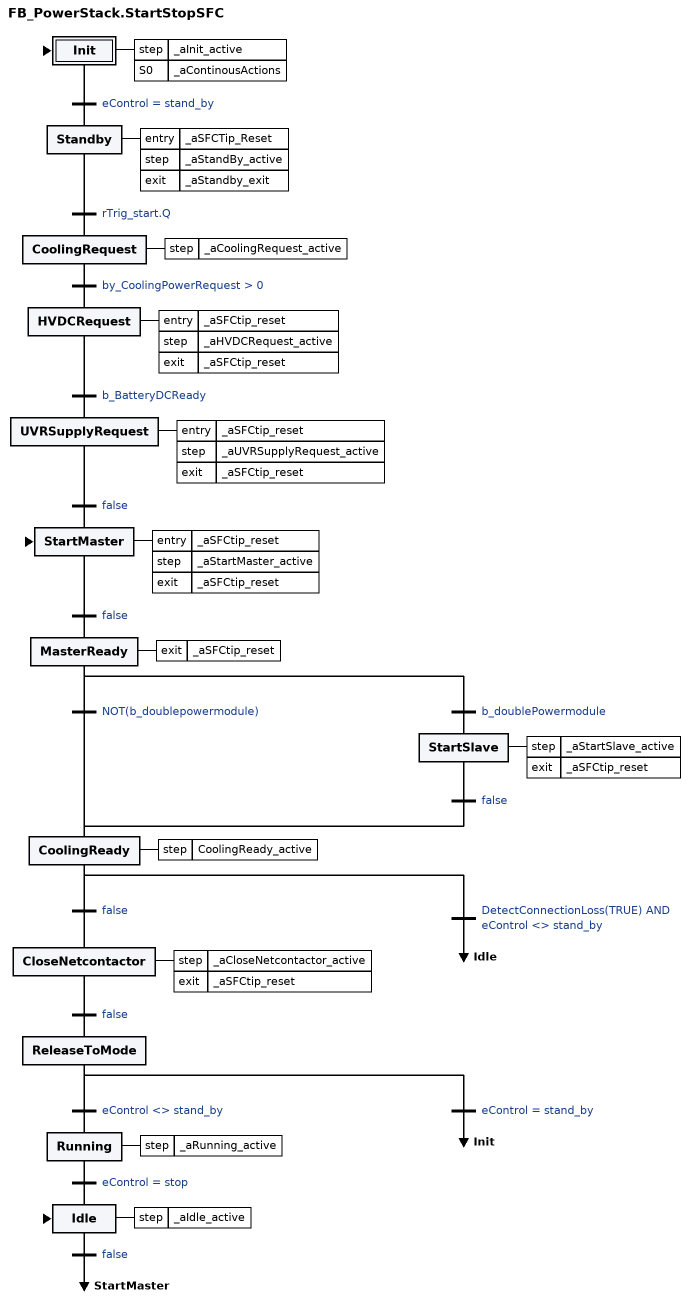
INITIAL_STEP Init:
    _aInit_active(N);  // step action
    _aContinousActions(S0);
END_STEP
TRANSITION FROM Init TO Standby
    := eControl = stand_by;
END_TRANSITION
STEP Standby:
    _aSFCTip_Reset(P1);  // entry action
    _aStandBy_active(N);  // step action
    _aStandby_exit(P0);  // exit action
END_STEP
TRANSITION FROM Standby TO CoolingRequest
    := rTrig_start.Q;
END_TRANSITION
STEP CoolingRequest:  // max time T#30s
    _aCoolingRequest_active(N);  // step action
END_STEP
TRANSITION FROM CoolingRequest TO HVDCRequest
    := by_CoolingPowerRequest > 0;
END_TRANSITION
STEP HVDCRequest:  // max time T#30s
    _aSFCtip_reset(P1);  // entry action
    _aHVDCRequest_active(N);  // step action
    _aSFCtip_reset(P0);  // exit action
END_STEP
TRANSITION FROM HVDCRequest TO UVRSupplyRequest
    := b_BatteryDCReady;
END_TRANSITION
STEP UVRSupplyRequest:  // max time T#30s
    _aSFCtip_reset(P1);  // entry action
    _aUVRSupplyRequest_active(N);  // step action
    _aSFCtip_reset(P0);  // exit action
END_STEP
TRANSITION FROM UVRSupplyRequest TO StartMaster
    := false;
END_TRANSITION
STEP StartMaster:  // min time T#1s
    _aSFCtip_reset(P1);  // entry action
    _aStartMaster_active(N);  // step action
    _aSFCtip_reset(P0);  // exit action
END_STEP
TRANSITION FROM StartMaster TO MasterReady
    := false;
END_TRANSITION
STEP MasterReady:  // min time T#1s
    _aSFCtip_reset(P0);  // exit action
END_STEP
TRANSITION FROM MasterReady TO CoolingReady
    := NOT(b_doublepowermodule);
END_TRANSITION
TRANSITION FROM MasterReady TO StartSlave
    := b_doublePowermodule;
END_TRANSITION
STEP StartSlave:  // max time T#30s
    _aStartSlave_active(N);  // step action
    _aSFCtip_reset(P0);  // exit action
END_STEP
TRANSITION FROM StartSlave TO CoolingReady
    := false;
END_TRANSITION
STEP CoolingReady:  // min time T#3s
    CoolingReady_active(N);  // step action
END_STEP
TRANSITION FROM CoolingReady TO CloseNetcontactor
    := false;
END_TRANSITION
STEP CloseNetcontactor:
    _aCloseNetcontactor_active(N);  // step action
    _aSFCtip_reset(P0);  // exit action
END_STEP
TRANSITION FROM CloseNetcontactor TO ReleaseToMode
    := false;
END_TRANSITION
TRANSITION FROM CoolingReady TO Idle
    := DetectConnectionLoss(TRUE) AND eControl <> stand_by;
END_TRANSITION
STEP ReleaseToMode:  // min time T#10ms
END_STEP
TRANSITION FROM ReleaseToMode TO Running
    := eControl <> stand_by;
END_TRANSITION
STEP Running:  // min time T#50ms
    _aRunning_active(N);  // step action
END_STEP
TRANSITION FROM Running TO Idle
    := eControl = stop;
END_TRANSITION
TRANSITION FROM ReleaseToMode TO Init
    := eControl = stand_by;
END_TRANSITION
STEP Idle:  // min time T#500ms
    _aIdle_active(N);  // step action
END_STEP
TRANSITION FROM Idle TO StartMaster
    := false;
END_TRANSITION
// branch label Branch5_StartStopSFC
// branch label Branch7_StartStopSFC
// branch label Branch6_StartStopSFC
END_ACTION

METHOD Stopcmd : BOOL
IF NOT(get.e_State = eStatusPowerstack.fault) THEN
	eControl := Stop;
END_IF

//if SFC transition occurs, give feedback.
Stopcmd := get.e_State = eStatusPowerStack.idle;
END_METHOD

END_FUNCTION_BLOCK

// ---- POUs/Objects/PowerStack/NetContactor/FB_NetContactor.TcPOU
FUNCTION_BLOCK FB_NetContactor
VAR_OUTPUT
	get								: ST_Netcontactor_get;
	b_NetcontEDM					: BOOL;
END_VAR 

VAR_INPUT
	set								: ST_Netcontactor_set;
END_VAR

VAR
	IO								: FB_NetContactor_IO;
	events							: st_Netcontactor_events;
	b_reset							: BOOL;
	ton_ForceCloseDelay				: TON := (PT := T#500MS);
	fTrigForceCloseReset			: F_TRIG;
END_VAR

io(b_RotationSelect := SetRotationSwitch(), get:=get, b_NetcontEDM:=b_NetcontEDM);
get.b_NetConFb := get.b_NetcontRightFb OR get.b_NetcontLeftFb;

//close delay + reset mechanism. Required for AC detection prior to the force being instaniously executed.
ton_ForceCloseDelay();
fTrigForceCloseReset(CLK := get.b_NetConFb);
IF fTrigForceCloseReset.Q THEN
	ton_ForceCloseDelay.IN := FALSE;
END_IF

IF get.b_NetConFb AND io.b_ForceCloseCommand THEN
	get.b_SyncCloseCommand := FALSE;
END_IF


//Converter netcontactor control mode to open/close request
CheckFeedback(get:= get, b_NetconFbRight := get.b_NetcontRightFb, b_NetConFbLeft := get.b_NetcontLeftFb);

METHOD PRIVATE CheckFeedback : BOOL
VAR
	ton_MaxTime					: TON;
END_VAR

VAR_IN_OUT
	get							: ST_Netcontactor_get;
END_VAR

VAR_IN_OUT CONSTANT
		b_NetConFbLeft				: BOOL;
		b_NetConFbRight				: BOOL;	
END_VAR

VAR_INST
	sr_LeftfbFault				: SR;
	sr_rightfbFault				: SR;
	sr_fbTimeout				: SR;
END_VAR
get.events.b_ContactorLeftFbFault := FALSE;
get.events.b_ContactorRightFbFault := FALSE;

ton_MaxTime();

//SET Sync or force time-out
IF get.b_SyncCloseCommand THEN //long evaluation time if sync required
	ton_MaxTime.IN := TRUE;
	ton_MaxTime.PT := T#10S;
ELSIF io.b_ForceCloseCommand THEN  //shorter evaluation time if force required
	ton_MaxTime.IN := TRUE;
	ton_MaxTime.PT := T#1S;
ELSE
	ton_MaxTime.IN:= FALSE;
END_IF

//set diagnostics + Feedback signal accordingly
sr_LeftfbFault(SET1 	:= NOT(b_NetConFbLeft) AND ton_MaxTime.Q AND io.b_RotationSelect,
			RESET 		:= b_reset,
			Q1			=> get.events.b_ContactorLeftFbFault); 	
sr_rightfbFault(SET1 	:= NOT(b_NetConFbRight) AND ton_MaxTime.Q AND NOT io.b_RotationSelect,
			RESET 		:= b_reset,
			Q1			=> get.events.b_ContactorLeftFbFault);	


			
sr_FbTimeout(SET1:= ton_MaxTime.Q, RESET :=b_reset, Q1 => get.events.b_ContactorFbTimeout);		
//Set output to external program
IF b_NetConFbLeft THEN
	get.e_NetConState := eNetcontactorstate.LeftClosed;
ELSIF b_NetConFbRight THEN
	get.e_NetConState := eNetcontactorstate.RightClosed;
ELSE
	get.e_NetConState := eNetcontactorstate.open;
END_IF
END_METHOD

METHOD Close : BOOL;
VAR_INPUT
	b_force	: BOOL;
END_VAR



VAR_INST
	tof_ReleaseForce : TOF := (PT := T#0S);
END_VAR


IF set.e_ClosingRequest <>  eNetcontMode.none THEN
	IF NOT Settings.Configuration.b_AutomaticACrotation AND set.e_ClosingRequest = eNetcontMode.left THEN //if left is requested without this option, don't close the netcontactor.
		b_Force := FALSE;
		get.b_SyncCloseCommand := FALSE;
		get.events.b_IllegalLeftFieldSelected := TRUE;
	ELSE
		get.events.b_IllegalLeftFieldSelected := FALSE;
		ton_ForceCloseDelay.IN := b_Force;
		// IF not already closed
		IF ton_ForceCloseDelay.Q THEN 
			tof_ReleaseForce(IN := TRUE);						//Enable force in AND..
			get.b_SyncCloseCommand := FALSE; 		//Avoid sending sync command simultaniously
		ELSE
			tof_ReleaseForce(IN := FALSE);
			get.b_SyncCloseCommand := TRUE;
		END_IF
		
		//To avoid instatanous forcing in when sync should have been done from initial start to grid sync,
		IF NOT get.b_NetConFb THEN
			io.b_ForceCloseCommand :=  NOT get.b_SyncCloseCommand;
		ELSE
			io.b_ForceCloseCommand := tof_ReleaseForce.Q OR get.b_NetConFb;
		END_IF
	END_IF
END_IF

Close := get.b_NetConFb; // io.b_ForceCloseCommand <> get.b_SyncCloseCommand AND
END_METHOD

METHOD GetDiagnostics
VAR_IN_OUT
	AddError		: ARRAY [*] OF FB_AddErrorST;
	a_ActiveEvents	: ARRAY [*] OF ST_ErrorStruct;
	w_Index			: WORD;
END_VAR
	(*Right fb fault*)		AddError[w_Index](
					b_ErrorTrig			:= get.events.b_ContactorRightFbFault,
					out_ST_Error			:= a_ActiveEvents[w_Index],
					w_ErrorID					:= 1,
					e_ObjectID				:= eObject_ID.Netcontactor,
					s_Message				:= 'right feedback fault',
					e_sev					:= eSeverity.NormalShutdown
				);
				w_Index := w_Index +1;
		
	(*left fb fault*)		AddError[w_Index](
					b_ErrorTrig			:= get.events.b_ContactorleftFbFault,
					out_ST_Error			:= a_ActiveEvents[w_Index],
					w_ErrorID					:= 2,
					s_Message				:= 'left feedback fault',
					e_sev					:= eSeverity.NormalShutdown
				);
				w_Index := w_Index +1;
		
	(*Phase Rotation fault*)			AddError[w_Index](
					b_ErrorTrig				:= get.events.b_PhaseRotationFault,
					out_ST_Error			:= a_ActiveEvents[w_Index],
					w_ErrorID				:= 3,
					s_Message				:= 'Phase rotation fault detected',
					e_sev					:= eSeverity.quickshutdown,
					b_AutoClear				:= TRUE
				);
				w_Index := w_Index +1;

	(*wrong Rotation selected fault*)			AddError[w_Index](
					b_ErrorTrig				:= get.events.b_IllegalLeftFieldSelected,
					out_ST_Error			:= a_ActiveEvents[w_Index],
					w_ErrorID				:= 4,
					s_Message				:= 'Left rotating field selected while not available',
					e_sev					:= eSeverity.Warning,
					b_AutoClear				:= TRUE
				);
				w_Index := w_Index +1;
END_METHOD

METHOD Open : BOOL

VAR_INST
	//ton_delay			: TON := (PT:= T#1S);
END_VAR
//ton_delay(IN:=get.b_NetConFb);

io.b_ForceCloseCommand := FALSE;
get.b_SyncCloseCommand := FALSE;
ton_ForceCloseDelay.IN := get.b_NetConFb;

open := NOT get.b_NetConFb;
END_METHOD

METHOD Reset : BOOL
b_reset := TRUE;

IF NOT get.events.b_ContactorFbTimeout OR NOT get.events.b_ContactorLeftFbFault OR NOT get.events.b_ContactorRightFbFault THEN;
	b_reset := FALSE;
	reset := TRUE;
END_IF
END_METHOD

METHOD SetEvents : BOOL
VAR_INPUT
END_VAR
//Phase rotation fault
get.events.b_PhaseRotationFault := set.e_ACRotationState = eACRotationState.Left AND NOT set.b_RotationSwitchEnable;
END_METHOD

METHOD PRIVATE SetRotationSwitch : BOOL

VAR_INST
	RotationLeft			: BOOL;
END_VAR
IF NOT get.b_NetConFb THEN
	IF Settings.Configuration.b_AutomaticACrotation THEN //only when option is available.
		CASE set.e_ACRotationState OF
			0: //NO ac
			CASE set.e_ClosingRequest OF
				eNetcontMode.right: RotationLeft := 0;
				eNetcontMode.left: RotationLeft := 1;
				eNetcontMode.auto: RotationLeft := 0;
			END_CASE
			1: RotationLeft := 0;
			-1: RotationLeft := 1;
		END_CASE
	ELSE
			RotationLeft := 0;
	END_IF
END_IF

SetRotationSwitch := RotationLeft;
END_METHOD

END_FUNCTION_BLOCK

// ---- POUs/Objects/PowerStack/NetContactor/FB_NetContactor_IO.TcPOU
FUNCTION_BLOCK FB_NetContactor_IO
VAR
	b_Write					AT %Q* : ARRAY[1..2] OF BOOL;	
	b_Read					AT %I* : ARRAY[1..3] OF BOOL;
END_VAR

VAR_INPUT
	b_RotationSelect					: BOOL := 0; //0: Clockwise, 1: Anti-Clockwise
	b_ForceCloseCommand					: BOOL := 0; //O; Open, 1:close
END_VAR

VAR_IN_OUT
	get								: ST_Netcontactor_get;
	b_NetcontEDM					: BOOL;
END_VAR
VAR
END_VAR

read();
Write();

METHOD PRIVATE Read
get.b_NetcontRightFb 	:= b_read[1];
get.b_NetcontLeftFb		:= b_read[2];
b_NetcontEDM			:= b_read[3];
END_METHOD

METHOD PRIVATE Write

VAR_INST
	
END_VAR
b_Write[1] := b_RotationSelect;
b_Write[2] := b_ForceCloseCommand;
END_METHOD

END_FUNCTION_BLOCK

// ---- POUs/Objects/PowerStack/PowerModule/FB_PowerModule.TcPOU
FUNCTION_BLOCK FB_PowerModule
VAR_IN_OUT CONSTANT
	st_params							: ST_PowerModule_params;
	st_calibration						: ST_PowerModule_Calibration;
END_VAR


VAR_INPUT
	set									: ST_PowerModule_set; //only setteable from intern powerstack function
	r_batteryDCVoltage					: REAL;
	b_enable							: BOOL;
	e_ID								: eObject_ID;
END_VAR

VAR_OUTPUT
	{attribute 'TcAnalytics'}
	get									: ST_PowerModule_get;
	b_MccbEDM							: BOOL;
END_VAR	

VAR									
	Inverter							: FB_PowerModule_Inverter();
	Buscoupler							: FB_PowerModule_Buscoupler();
	ton_ResetPulse						: TON := (PT:= T#100MS);
	
	r_Prq: REAL;
	r_Qrq: REAL;
	pin: REAL;
	QIN: REAL;
END_VAR

IF b_enable THEN
	get.b_online := get.ui_buscouplerCommStatus = 0 AND get.ui_InverterCommStatus = 0;
	
	//Instantiate function blocks
	Buscoupler(get:=get, b_MccbEDM := b_MccbEDM, b_D7SyncRq := set.b_D7SyncRequest);
	Inverter(set := set, get:=get, st_params:=st_params);
	//defaults
	Inverter.ControlWord.b_FieldbusControlEnable := st_params.b_FieldBusControlEnable;

	//Control fan contactor.
	FanControl(st_params := st_params);
	
	//Set PowerModule status
	GetPowerModuleStatus();
	
	//Set DroopLimit
	SetInverterSettings();
	
	//Calculate derivatives
	CalculateDerivativePowerValues();
	
	//Parallel Drive
	SetParallelDrive();
	
	//setEvents
	SetEvents(events := get.Events, st_params:=st_Params);
	
	//FILL GET STRUCT
	GetInverterModes();
	FillAdditionalGets(get, set);
	
	//inverter.ControlWord.b_Reset := FALSE;
	
	SetParallelDrive();
	
	IF get.StatusWord.b_Fault THEN
		Shutdown(TRUE);
	END_IF
	
	IF GVL.b_initCycle THEN
		init();
	END_IF
END_IF

r_Prq := CompensationCurve(PIN := pin, QIN := qin, coef := st_calibration.PCoefficients, mode := 0);
r_Qrq := CompensationCurve(PIN := pin, QIN := qin, coef := st_calibration.QCoefficients, mode := 1);

METHOD BaseValueToRef : REAL;
VAR_INPUT
	IN : REAL;
END_VAR
BaseValueToRef:= IN / MAX(1, st_params.r_InverterRatedCurrent) * 100;
END_METHOD

METHOD PRIVATE CalculateDerivativePowerValues : BOOL
get.r_ReactivePower	:= get.r_ACVoltageD7 * 1.73 * get.r_ReactiveCurrent / 1000; // kvar
get.r_ActivePower	:= get.r_ACVoltageSupply* 1.73 * get.r_activeCurrent / 1000;
get.r_ApparentPower	:= SQRT(MAX(0,EXPT(get.r_ActivePower,2) + EXPT(get.r_ReactivePower,2)));
get.r_LoadPercent	:= get.r_ACCurrent / MAX(1, st_params.r_InverterRatedCurrent) * 100;
get.r_DCPower		:= get.r_DCCurrent * get.r_DCVoltage / 1000; // kW
END_METHOD

METHOD CheckDCVoltage : BOOL

VAR_INST
	b_DCprechargeOK				: BOOL; 
	b_DCVoltageOK				: BOOL;
	ton_DCOKreleaseTime			: TON := (PT:= T#1S);
END_VAR
b_DCPrechargeOK := ABS(r_BatteryDCVoltage - get.r_DCVoltage) <=  st_params.ui_DCVoltageDeltaPrechargeOK;
b_DCVoltageOK := get.r_DCVoltage > st_params.ui_DCvoltageMinPrechargeOK;

ton_DCOKReleaseTime(IN:= b_DCPrechargeOK AND b_DCVoltageOK);

CheckDCVoltage :=ton_DCOKReleaseTime.Q;
END_METHOD

METHOD CompensationCurve : REAL
VAR_INPUT
	PIN			: REAL; 
	QIN			: REAL;
	mode		: BYTE; // 0 = Pout, 1 = Qout;
END_VAR

VAR_IN_OUT CONSTANT
	coef : ST_Powermodule_PowerCurveCoefficients;
END_VAR

VAR_INST
	Q1			: REAL;
	Q2			: REAL;
	disc 		: REAL;
	Avalues		: REAL;
	Bvalues		: REAL;
	Cvalues		: REAL;
	depVar		: REAL;
	indepVar	: REAL;
END_VAR
IF NOT coef.enable THEN
	CompensationCurve := SEL(mode =0, Qin, Pin);
	RETURN; // Geen reële oplossing
END_IF


IF mode = 0 THEN
	indepVar := Pin;
	depVar := Qin;

ELSE
	indepVar := Qin;
	depVar := Pin;
END_IF

Avalues := coef.a;
BValues := coef.c*depVar + coef.d;
CValues := coef.b*EXPT(depVar,2)+coef.e*depVar + coef.f - indepVar;

disc := EXPT(BValues,2)-(4*AValues*CValues);
IF disc < 0 THEN
	CompensationCurve := indepVar;
	RETURN; // Geen reële oplossing
END_IF

// Controleer discriminant
IF Avalues = 0 THEN
    // Lineaire oplossing: B * P + C = 0 → P = -C / B
    IF BValues = 0 THEN
        RETURN; // onoplosbaar
    ELSE
        CompensationCurve := -CValues / BValues;
        RETURN;
    END_IF
END_IF

// Kwadratische oplossing (ABC)
Q1 := (-BValues + SQRT(disc)) / (2 * Avalues);
Q2 := (-BValues - SQRT(disc)) / (2 * Avalues);
CompensationCurve := Q1;
//// Kies de beste wortel (voorbeeld: dichtsbijzijnde bij indepVar)
//IF ABS(Q1 - indepVar) < ABS(Q2 - indepVar) THEN
//    CompensationCurve := Q1;
//ELSE
//    CompensationCurve := Q2;
//END_IF
END_METHOD

METHOD PRIVATE CoupleDC : BOOL
VAR_INPUT
END_VAR
IF get.StatusWord.b_ReadyToDCCharge THEN
	buscoupler.b_DCprechargeContactor := TRUE;
	buscoupler.b_DCMainContactor := CheckDCvoltage();
	CoupleDC := get.b_DCcontactorFb;
END_IF
END_METHOD

METHOD PRIVATE DecoupleDC : BOOL

VAR_INST
	b_DCmainreleaseConditionOK 	:  BOOL;
	b_DCprereleaseConditionOK 	:  BOOL;
	ton_PrechargeReleaseDelay	:  TON := (PT:= T#1S);
END_VAR

VAR
	r_DCreleaseCurrent		: REAL := 5;
	r_DCreleaseVoltage		: REAL := 10;
END_VAR
// Release main contactor first based on current
b_DCmainreleaseConditionOK := ABS(get.r_DCCurrent) < r_DCreleaseCurrent AND NOT get.StatusWord.b_Running;
IF b_DCmainreleaseConditionOK THEN
	buscoupler.b_DCmainContactor := FALSE;
END_IF

// release precharge based on voltage contactor 
b_DCprereleaseConditionOK := NOT get.b_DCcontactorFb OR r_batteryDCVoltage < r_DCreleaseVoltage; //NOT get.b_DCcontactorFb (Not for units without precharge, rewire output4 to input 4 of buscoupler.)
ton_PrechargeReleaseDelay(IN:= b_DCprereleaseConditionOK); //some delay added to be sure
IF ton_PrechargeReleaseDelay.Q THEN
	buscoupler.b_DCprechargeContactor := FALSE;
END_IF 

//Give feedback
IF b_DCprereleaseConditionOK AND b_DCmainreleaseConditionOK THEN
	DecoupleDc := NOT buscoupler.b_DCprechargeContactor AND NOT get.b_DCcontactorFb;
END_IF
END_METHOD

METHOD PRIVATE FanControl : BOOL
VAR_IN_OUT CONSTANT
	st_params : ST_Powermodule_params;
END_VAR
	


VAR_INST
	b_fanOn				: BOOL;
	tof_FanOffDelay		: TOF := (PT := T#60S);
END_VAR
IF get.r_TemperatureMax > st_params.r_TempFanOn OR get.r_LoadPercent > st_params.r_powerLoadFanOn THEN
	b_fanOn := TRUE;
ELSIF get.r_TemperatureMax < st_params.r_TempFanOn - 5 AND get.r_LoadPercent < st_params.r_powerLoadFanOn - 10 THEN
	b_fanOn := FALSE;
END_IF


tof_FanOffDelay(
	IN:= b_fanOn);
	
buscoupler.b_FanOn := set.b_FanContactor OR tof_FanOffDelay.Q;
END_METHOD

METHOD FillAdditionalGets : BOOL
VAR_IN_OUT
		get : ST_Powermodule_get;
		set	: ST_Powermodule_set;
END_VAR
get.r_TemperatureMax := GetMaxTemperature();
get.r_Pset := set.r_ActivePower;
get.r_Qset := set.r_ReactivePower;
get.b_PrechargeContactor := buscoupler.b_DCprechargeContactor;
END_METHOD

METHOD GetDiagnostics 
VAR_IN_OUT
	AddError		: ARRAY [*] OF FB_AddErrorST;
	a_ActiveEvents	: ARRAY [*] OF ST_ErrorStruct;
	w_Index			: WORD;
END_VAR

VAR
	by_errCt	: BYTE;
	by_warnCt	: BYTE;
END_VAR


VAR_INST
	b_test: BOOL;
END_VAR
(*POWERMODULE*)
	//Inverter faults
	(*OverCurr Fault*)		AddError[w_Index](
			b_ErrorTrig			:= Get.Events.b_F1OverCurrent,
			out_ST_Error			:= a_ActiveEvents[w_Index],
			w_ErrorID					:= 1,
			e_objectID				:= e_ID,
			s_Message				:= 'overcurrent fault (F1)',
			e_sev					:= eSeverity.Quickshutdown,
			);
		IF AddError[w_Index].b_out THEN by_errCt := by_errCt + 1; END_IF;
		w_Index := w_Index +1;
		
	(*OverVolt Fault*)		AddError[w_Index](
			b_ErrorTrig			:= Get.Events.b_F2OverVoltage,
			out_ST_Error			:= a_ActiveEvents[w_Index],
			w_ErrorID					:= 2,
			s_Message				:= 'DC overvoltage fault (F2)',
			e_sev					:= eSeverity.Quickshutdown,
			);
		IF AddError[w_Index].b_out THEN by_errCt := by_errCt + 1; END_IF;
		w_Index := w_Index +1;
	
	(*UnderVolt Fault*)		AddError[w_Index](
			b_ErrorTrig			:= Get.Events.b_F9UnderVoltage,
			out_ST_Error			:= a_ActiveEvents[w_Index],
			w_ErrorID					:= 3,
			s_Message				:= 'DC undervoltage fault (F9)',
			e_sev					:= eSeverity.Quickshutdown,
			);
		IF AddError[w_Index].b_out THEN by_errCt := by_errCt + 1; END_IF;
		w_Index := w_Index +1;
	
	(*ShortCurr Fault*)		AddError[w_Index](
			b_ErrorTrig		:= Get.Events.b_F91ShortCircuit,
			out_ST_Error			:= a_ActiveEvents[w_Index],
			w_ErrorID					:= 4,
			s_Message				:= 'short circuit fault (F91)',
			e_sev					:= eSeverity.Quickshutdown,
			);
		IF AddError[w_Index].b_out THEN by_errCt := by_errCt + 1; END_IF;
		w_Index := w_Index +1;
		
	(*Earth Fault*)			AddError[w_Index](
			b_ErrorTrig		:= Get.Events.b_F3EarthFault,
			out_ST_Error			:= a_ActiveEvents[w_Index],
			w_ErrorID					:= 5,
			s_Message				:= 'earth fault (F3)',
			e_sev					:= eSeverity.Quickshutdown,
			);
		IF AddError[w_Index].b_out THEN by_errCt := by_errCt + 1; END_IF;
		w_Index := w_Index +1;
		
	(*LineSync Fault*)		AddError[w_Index](
			b_ErrorTrig		:= Get.Events.b_F10LineSynchFault,
			out_ST_Error			:= a_ActiveEvents[w_Index],
			w_ErrorID					:= 6,
			s_Message				:= 'line synchronisation fault (F10)',
			e_sev					:= eSeverity.Quickshutdown,
			);
		IF AddError[w_Index].b_out THEN by_errCt := by_errCt + 1; END_IF;
		w_Index := w_Index +1;
	
	(*Keypad Fault*)		AddError[w_Index](
			b_ErrorTrig		:= Get.Events.b_F52KeypadOCCommFault,
			out_ST_Error			:= a_ActiveEvents[w_Index],
			w_ErrorID					:= 7,
			s_Message				:= 'keypad communication fault (F52)',
			e_sev					:= eSeverity.warning,
			);
		IF AddError[w_Index].b_out THEN by_errCt := by_errCt + 1; END_IF;
		w_Index := w_Index +1;
	
	(*Fieldbus Fault*)		AddError[w_Index](
			b_ErrorTrig		:= Get.Events.b_F53FieldbusFault,
			out_ST_Error			:= a_ActiveEvents[w_Index],
			w_ErrorID					:= 8,
			s_Message				:= 'fieldbus fault (F53)',
			e_sev					:= eSeverity.Quickshutdown,
			);
		IF AddError[w_Index].b_out THEN by_errCt := by_errCt + 1; END_IF;
		w_Index := w_Index +1;
		
	(*Systembus Fault*)		AddError[w_Index](
			b_ErrorTrig		:= Get.Events.b_F59SystembusFault,
			out_ST_Error			:= a_ActiveEvents[w_Index],
			w_ErrorID					:= 9,
			s_Message				:= 'system bus Fault (F59)',
			e_sev					:= eSeverity.Quickshutdown,
			);
		IF AddError[w_Index].b_out THEN by_errCt := by_errCt + 1; END_IF;
		w_Index := w_Index +1;
	
	(*IOslot Fault*)		AddError[w_Index](
			b_ErrorTrig		:= Get.Events.b_F54SlotCommunicationFault,
			out_ST_Error			:= a_ActiveEvents[w_Index],
			w_ErrorID					:= 10,
			s_Message				:= 'IO slot communication fault (F54)',
			e_sev					:= eSeverity.Quickshutdown,
			);
		IF AddError[w_Index].b_out THEN by_errCt := by_errCt + 1; END_IF;
		w_Index := w_Index +1;
		
	(*4ma meas Fault*)		AddError[w_Index](
			b_ErrorTrig		:= Get.Events.b_F50Meas4mAFault,
			out_ST_Error			:= a_ActiveEvents[w_Index],
			w_ErrorID					:= 11,
			s_Message				:= 'measurement 4 mA fault (F50)',
			e_sev					:= eSeverity.info,
			b_AutoClear			:= TRUE,
		);
		w_Index := w_Index +1;
		
	(*Watchdog Fault*)		AddError[w_Index](
			b_ErrorTrig		:= Get.Events.b_WatchdogError,
			out_ST_Error			:= a_ActiveEvents[w_Index],
			w_ErrorID					:= 12,
			s_Message				:= 'watchdog fault',
			e_sev					:= eSeverity.Quickshutdown,
			);
		IF AddError[w_Index].b_out THEN by_errCt := by_errCt + 1; END_IF;
		w_Index := w_Index +1;
	
	(*Mccb Trip*)			AddError[w_Index](
			b_ErrorTrig			:= FALSE, //Get.Events.b_MCCBtrip,
			out_ST_Error			:= a_ActiveEvents[w_Index],
			w_ErrorID					:= 13,
			s_Message				:= 'MCCB trip',
			e_sev					:= eSeverity.warning
		);
		w_Index := w_Index +1;

	(*Shutdown TimeOut*)			AddError[w_Index](
			b_ErrorTrig			:= Get.Events.b_ShutdownTimeOut,
			out_ST_Error			:= a_ActiveEvents[w_Index],
			w_ErrorID					:= 14,
			s_Message				:= 'shutdown Timeout',
			e_sev					:= eSeverity.QuickShutdown
		);
		w_Index := w_Index +1;
		
	(*output phase fault (F11)*)	AddError[w_Index](
			b_ErrorTrig				:= Get.Events.b_F11OutputPhaseFault,
			out_ST_Error			:= a_ActiveEvents[w_Index],
			w_ErrorID				:= 15,
			s_Message				:= 'output phase fault (F11)',
			e_sev					:= eSeverity.Quickshutdown
		);
		w_Index := w_Index +1;
		
	(*charge fault (F80)*)			AddError[w_Index](
			b_ErrorTrig				:= Get.Events.b_F80ChargeFault,
			out_ST_Error			:= a_ActiveEvents[w_Index],
			w_ErrorID				:= 16,
			s_Message				:= 'charge fault (F80)',
			e_sev					:= eSeverity.Quickshutdown
		);
		w_Index := w_Index +1;
		
		(*charge fault (F80)*)			AddError[w_Index](
			b_ErrorTrig				:= Get.Events.b_F51ExternalFault,
			out_ST_Error			:= a_ActiveEvents[w_Index],
			w_ErrorID				:= 17,
			s_Message				:= 'external fault (F51)',
			e_sev					:= eSeverity.Quickshutdown
		);
		w_Index := w_Index +1;
		
		(*IGBT fault (F31)*)		AddError[w_Index](
			b_ErrorTrig				:= Get.Events.b_F31IGBTFault,
			out_ST_Error			:= a_ActiveEvents[w_Index],
			w_ErrorID				:= 18,
			s_Message				:= 'IGBT fault (F31)',
			e_sev					:= eSeverity.Quickshutdown
		);
		w_Index := w_Index +1;
		
		(*MCB state fault (F64)*)		AddError[w_Index](
			b_ErrorTrig				:= Get.Events.b_F64MCBstateFault,
			out_ST_Error			:= a_ActiveEvents[w_Index],
			w_ErrorID				:= 19,
			s_Message				:= 'MCB state fault (F64)',
			e_sev					:= eSeverity.Quickshutdown
		);
		w_Index := w_Index +1;
	
	//Temperature Faults
	(*Gridch L1 Alarm*)		AddError[w_Index](
			b_ErrorTrig		:= Get.Events.b_CMChokeTemperatureTooHigh[1],
			out_ST_Error			:= a_ActiveEvents[w_Index],
			w_ErrorID					:= 20 ,
			s_Message				:= 'gridchoke L1 temperature too high',
			e_sev					:= eSeverity.normalshutdown,
			);
		IF AddError[w_Index].b_out THEN by_errCt := by_errCt + 1; END_IF;
		w_Index := w_Index +1;
		
	(*Gridch L2 Alarm*)		AddError[w_Index](
			b_ErrorTrig		:= Get.Events.b_CMChokeTemperatureTooHigh[2], //phase 2
			out_ST_Error			:= a_ActiveEvents[w_Index],
			w_ErrorID					:= 21 ,
			s_Message				:= 'gridchoke L2 temperature too high',
			e_sev					:= eSeverity.normalshutdown,
			);
		IF AddError[w_Index].b_out THEN by_errCt := by_errCt + 1; END_IF;
		w_Index := w_Index +1;
		
	(*Gridch L3 Alarm*)		AddError[w_Index](
			b_ErrorTrig		:= Get.Events.b_CMChokeTemperatureTooHigh[3], //phase 3
			out_ST_Error			:= a_ActiveEvents[w_Index],
			w_ErrorID					:= 22 ,
			s_Message				:= 'gridchoke L3 temperature too high',
			e_sev					:= eSeverity.normalshutdown,
			);
		IF AddError[w_Index].b_out THEN by_errCt := by_errCt + 1; END_IF;
		w_Index := w_Index +1;
		
	(*CMch L1 Alarm*)		AddError[w_Index](
			b_ErrorTrig		:= Get.Events.b_GridChokeTemperatureTooHigh[1], //phase 1
			out_ST_Error			:= a_ActiveEvents[w_Index],
			w_ErrorID					:= 23 ,
			s_Message				:= 'CM choke L1 temperature too high',
			e_sev					:= eSeverity.normalshutdown,
			);
		IF AddError[w_Index].b_out THEN by_errCt := by_errCt + 1; END_IF;
		w_Index := w_Index +1;
		
	(*CMch L2 Alarm*)		AddError[w_Index](
			b_ErrorTrig		:= Get.Events.b_CMChokeTemperatureTooHigh[2], //phase 2
			out_ST_Error			:= a_ActiveEvents[w_Index],
			w_ErrorID					:= 24 ,
			s_Message				:= 'CM choke L2 temperature too high',
			e_sev					:= eSeverity.normalshutdown,
			);
		IF AddError[w_Index].b_out THEN by_errCt := by_errCt + 1; END_IF;
		w_Index := w_Index +1;
		
	(*CMch L3 Alarm*)		AddError[w_Index](
			b_ErrorTrig		:= Get.Events.b_CMChokeTemperatureTooHigh[3], //phase 3
			out_ST_Error			:= a_ActiveEvents[w_Index],
			w_ErrorID					:= 25 ,
			s_Message				:= 'CM choke L3 temperature too high',
			e_sev					:= eSeverity.normalshutdown,
			);
		IF AddError[w_Index].b_out THEN by_errCt := by_errCt + 1; END_IF;
		w_Index := w_Index +1;
		
	(*CMch DC Alarm*)		AddError[w_Index](
			b_ErrorTrig		:= Get.Events.b_CMChokeTemperatureTooHigh[4], //DC
			out_ST_Error			:= a_ActiveEvents[w_Index],
			w_ErrorID					:= 26 ,
			s_Message				:= 'CM choke DC temperature too high',
			e_sev					:= eSeverity.normalshutdown,
			);
		IF AddError[w_Index].b_out THEN by_errCt := by_errCt + 1; END_IF;
		w_Index := w_Index +1;
		
	(*Inverter Alarm*)		AddError[w_Index](
			b_ErrorTrig		:= Get.Events.b_F14UnitOverTemperature,
			out_ST_Error			:= a_ActiveEvents[w_Index],
			w_ErrorID					:= 27 ,
			s_Message				:= 'overtemperature fault (F14)',
			e_sev					:= eSeverity.Quickshutdown
		);
		IF AddError[w_Index].b_out THEN by_errCt := by_errCt + 1; END_IF;
		w_Index := w_Index +1;	
		
	(*PT100 Fault*)			AddError[w_Index](
			b_ErrorTrig		:= Get.Events.b_F56TemperatureFault, //inverter Pt100 measurement
			out_ST_Error			:= a_ActiveEvents[w_Index],
			w_ErrorID					:= 28 ,
			s_Message				:= 'pt100 temperature fault (F56)',
			e_sev					:= eSeverity.normalshutdown,
			);
		IF AddError[w_Index].b_out THEN by_errCt := by_errCt + 1; END_IF;
		w_Index := w_Index +1;
		
	
	//Temperature Warnings
	(*Gridch L1 Warning*)	AddError[w_Index](
			b_ErrorTrig			:= Get.Events.b_gridChokeTemperatureHigh[1], //phase 1
			out_ST_Error			:= a_ActiveEvents[w_Index],
			w_ErrorID					:= 40 ,
			s_Message				:= 'gridchoke L1 temperature high',
			e_sev					:= eSeverity.warning,
			b_AutoClear			:= TRUE,
			);
		IF AddError[w_Index].b_out THEN by_warnCt := by_warnCt + 1; END_IF;
		w_Index := w_Index +1;
		
	(*Gridch L2 Warning*)	AddError[w_Index](
			b_ErrorTrig		:= Get.Events.b_GridchokeTemperatureHigh[2], //phase 2
			out_ST_Error			:= a_ActiveEvents[w_Index],
			w_ErrorID					:= 41 ,
			s_Message				:= 'gridchoke L2 temperature high',
			e_sev					:= eSeverity.warning,
			b_AutoClear			:= TRUE,
			);
		IF AddError[w_Index].b_out THEN by_warnCt := by_warnCt + 1; END_IF;
		w_Index := w_Index +1;
		
	(*Gridch L3 Warning*)	AddError[w_Index](
			b_ErrorTrig		:= Get.Events.b_GridChokeTemperatureHigh[3], //phase 3
			out_ST_Error			:= a_ActiveEvents[w_Index],
			w_ErrorID					:= 42 ,
			s_Message				:= 'gridchoke L3 temperature high',
			e_sev					:= eSeverity.warning,
			b_AutoClear			:= TRUE,
			);
		IF AddError[w_Index].b_out THEN by_warnCt := by_warnCt + 1; END_IF;
		w_Index := w_Index +1;
		
	(*CMch L1 Warning*)		AddError[w_Index](
			b_ErrorTrig		:= Get.Events.b_CMChokeTemperatureHigh[1], //phase 1
			out_ST_Error			:= a_ActiveEvents[w_Index],
			w_ErrorID					:= 43 ,
			s_Message				:= 'CM choke L1 temperature high',
			e_sev					:= eSeverity.warning,
			b_AutoClear			:= TRUE,
			);
		IF AddError[w_Index].b_out THEN by_warnCt := by_warnCt + 1; END_IF;
		w_Index := w_Index +1;
		
	(*CMch L2 Warning*)		AddError[w_Index](
			b_ErrorTrig		:= Get.Events.b_CMChokeTemperatureHigh[2], //phase 2
			out_ST_Error			:= a_ActiveEvents[w_Index],
			w_ErrorID				:= 44 ,
			s_Message				:= 'CM choke L2 temperature high',
			e_sev					:= eSeverity.warning,
			b_AutoClear			:= TRUE,
			);
		IF AddError[w_Index].b_out THEN by_warnCt := by_warnCt + 1; END_IF;
		w_Index := w_Index +1;
		
	(*CMch L3 Warning*)		AddError[w_Index](
			b_ErrorTrig		:= Get.Events.b_CMChokeTemperatureHigh[3], //phase 3
			out_ST_Error			:= a_ActiveEvents[w_Index],
			w_ErrorID					:= 45 ,
			s_Message				:= 'CM choke L3 temperature high',
			e_sev					:= eSeverity.warning,
			b_AutoClear			:= TRUE,
			);
		IF AddError[w_Index].b_out THEN by_warnCt := by_warnCt + 1; END_IF;
		w_Index := w_Index +1;
		
	(*CMch DC Warning*)		AddError[w_Index](
			b_ErrorTrig		:= Get.Events.b_CMChokeTemperatureHigh[4], //DC
			out_ST_Error			:= a_ActiveEvents[w_Index],
			w_ErrorID					:= 46 ,
			s_Message				:= 'CM choke DC temperature high',
			e_sev					:= eSeverity.warning,
			b_AutoClear			:= TRUE,
			);
		IF AddError[w_Index].b_out THEN by_warnCt := by_warnCt + 1; END_IF;
		w_Index := w_Index +1;
		
	(*Inverter Warning*)	AddError[w_Index](
			b_ErrorTrig			:= Get.Events.b_inverterTemperatureHigh, //inverter
			out_ST_Error			:= a_ActiveEvents[w_Index],
			w_ErrorID					:= 47 ,
			s_Message				:= 'Inverter temperature high',
			e_sev					:= eSeverity.warning,
			b_AutoClear			:= TRUE,
			);
		IF AddError[w_Index].b_out THEN by_warnCt := by_warnCt + 1; END_IF;
		w_Index := w_Index +1;
		
	(*PT100 Range Warning*)	AddError[w_Index](
			b_ErrorTrig			:= Get.Events.b_CMSTemperatureRangeWarning, //inverter Pt100 measurement
			out_ST_Error			:= a_ActiveEvents[w_Index],
			w_ErrorID					:= 48 ,
			s_Message				:= 'CMS pt100 temperature range warning',
			e_sev					:= eSeverity.warning,
			b_AutoClear			:= TRUE,
			);
		IF AddError[w_Index].b_out THEN by_warnCt := by_warnCt + 1; END_IF;
		w_Index := w_Index +1;
		
	(*FanState Warning*)	AddError[w_Index](
			b_ErrorTrig			:= Get.Events.b_FanStateUnknownWarning, //general warning from inverter
			out_ST_Error			:= a_ActiveEvents[w_Index],
			w_ErrorID					:= 61 ,
			s_Message				:= 'fan state warning',
			e_sev					:= eSeverity.warning,
			t_triggerTime			:= T#1S,
			b_AutoClear				:= TRUE,
			);
		IF AddError[w_Index].b_out THEN by_warnCt := by_warnCt + 1; END_IF;
		w_Index := w_Index +1;
	
	(*PT100Underrange*)	AddError[w_Index](
			b_ErrorTrig			:= Get.Events.b_PT100Underrange, //general warning from inverter
			out_ST_Error			:= a_ActiveEvents[w_Index],
			w_ErrorID					:= 62 ,
			s_Message				:= 'PT100 underrange warning',
			e_sev					:= eSeverity.warning,
			b_AutoClear			:= TRUE,
			);
		IF AddError[w_Index].b_out THEN by_warnCt := by_warnCt + 1; END_IF;
		w_Index := w_Index +1;
		
	(*PT100Overrange*)	AddError[w_Index](
			b_ErrorTrig			:= Get.Events.b_PT100Underrange, //general warning from inverter
			out_ST_Error			:= a_ActiveEvents[w_Index],
			w_ErrorID					:= 63 ,
			s_Message				:= 'PT100 Overrange warning',
			e_sev					:= eSeverity.warning,
			b_AutoClear			:= TRUE,
			);
		IF AddError[w_Index].b_out THEN by_warnCt := by_warnCt + 1; END_IF;
		w_Index := w_Index +1;

	(*PT100 Error*)	AddError[w_Index](
			b_ErrorTrig			:= Get.Events.by_PT100ErrorCount > 5, //general warning from inverter
			out_ST_Error			:= a_ActiveEvents[w_Index],
			w_ErrorID					:= 64 ,
			s_Message				:= 'more than 5 PT100 errors',
			e_sev					:= eSeverity.Normalshutdown,
			b_AutoClear			:= TRUE,
			);
		IF AddError[w_Index].b_out THEN by_errCt := by_errCt + 1; END_IF;
		w_Index := w_Index +1;
		
	(*Buscoupler comm error*)	AddError[w_Index](
			b_ErrorTrig			:= Get.ui_BuscouplerCommStatus <>0, //general warning from inverter
			out_ST_Error			:= a_ActiveEvents[w_Index],
			w_ErrorID					:= 65 ,
			s_Message				:= 'buscoupler communication error',
			e_sev					:= eSeverity.Normalshutdown,
			);
		IF AddError[w_Index].b_out THEN by_errCt := by_errCt + 1; END_IF;
		w_Index := w_Index +1;
	
	(*Inverter comm error*)	AddError[w_Index](
			b_ErrorTrig			:= Get.ui_InverterCommStatus <>0 AND Get.ui_InverterCommStatus <15, //general warning from inverter
			out_ST_Error			:= a_ActiveEvents[w_Index],
			w_ErrorID					:= 66 ,
			s_Message				:= 'inverter communication error',
			e_sev					:= eSeverity.Quickshutdown
			);
		IF AddError[w_Index].b_out THEN by_errCt := by_errCt + 1; END_IF;
		w_Index := w_Index +1;
		
	(*Inverter temp throttling active*)	AddError[w_Index](
			b_ErrorTrig			:= get.Events.b_TempThrottlingActive, //general warning from inverter
			out_ST_Error			:= a_ActiveEvents[w_Index],
			w_ErrorID					:= 67 ,
			s_Message				:= 'temperature throttling active',
			e_sev					:= eSeverity.Warning,
			b_AutoClear			:= TRUE,
			);
		IF AddError[w_Index].b_out THEN by_warnCt := by_warnCt + 1; END_IF;
		w_Index := w_Index +1;
		
	(*Inverter current throttling active*)	AddError[w_Index](
			b_ErrorTrig			:= get.Events.b_CurrThrottlingActive, //general warning from inverter
			out_ST_Error			:= a_ActiveEvents[w_Index],
			w_ErrorID					:= 68 ,
			s_Message				:= 'Current throttling active',
			e_sev					:= eSeverity.Warning,
			b_AutoClear			:= TRUE,
			);
		IF AddError[w_Index].b_out THEN by_warnCt := by_warnCt + 1; END_IF;
		w_Index := w_Index +1;
		
		(*Inverter current throttling active*)	AddError[w_Index](
			b_ErrorTrig			:= get.StatusWord.b_Fault, //general warning from inverter
			out_ST_Error			:= a_ActiveEvents[w_Index],
			w_ErrorID					:= 69,
			s_Message				:= 'General fault',
			e_sev					:= eSeverity.Quickshutdown,
			);
		IF AddError[w_Index].b_out THEN by_errCt := by_errCt + 1; END_IF;
		w_Index := w_Index +1;
		
		(*UVR fault*)			AddError[w_Index](
			b_ErrorTrig				:= Get.Events.b_24VdcUVRFault,
			out_ST_Error			:= a_ActiveEvents[w_Index],
			w_ErrorID				:= 70,
			s_Message				:= 'UVR 24VDC Fault',
			e_sev					:= eSeverity.warning,
			b_AutoClear				:= TRUE,
		);
		w_Index := w_Index +1;

			

get.events.b_GeneralFaultFlag := by_errCt <> 0;
get.events.b_GeneralWarningFlag := by_warnCt <>0;
END_METHOD

METHOD PRIVATE GetInverterModes
IF get.UgridStatusWord.b_AFEmodeActive THEN
	get.e_InverterMode := eInvertermodes.afe;
ELSIF get.UgridStatusWord.b_IslandModeActive OR get.UgridStatusWord.b_MicrogridModeActive AND get.r_FrequencyDroop <= 0.1 THEN
	get.e_InverterMode := eInvertermodes.Island;	
ELSE
	get.e_InverterMode := eInvertermodes.Microgrid;
END_IF
END_METHOD

METHOD PRIVATE GetMaxTemperature : REAL;
// calculate max
GetMaxTemperature := MAX(
						get.r_TemperatureCMChoke[1], 
						get.r_TemperatureCMChoke[2], 
						get.r_TemperatureCMChoke[3], 
						get.r_TemperatureCMChoke[4],
						get.r_TemperatureGridChoke[1], 
						get.r_TemperatureGridChoke[2], 
						get.r_TemperatureGridChoke[3]
);
END_METHOD

METHOD PRIVATE GetPowerModuleStatus : BOOL
IF get.StatusWord.b_Fault OR get.Events.b_GeneralFaultFlag THEN
	get.e_Status := eStatusPowerModule.fault;
ELSIF get.StatusWord.b_Running THEN
	get.e_Status := eStatusPowermodule.running;
ELSIF get.StatusWord.b_ReadyToOperate THEN
	get.e_Status := eStatusPowermodule.idle;
ELSIF get.StatusWord.b_DCAtReference THEN	
	get.e_Status := eStatusPowermodule.DcOK;
ELSIF get.StatusWord.b_ReadyToDCCharge THEN
	get.e_Status := eStatusPowermodule.off;
ELSE
	get.e_Status := eStatusPowermodule.Init;
END_IF
END_METHOD

METHOD GetTemperatureEvents : BOOL
VAR_INPUT
	Warnings	: 	BOOL;
END_VAR
IF Warnings THEN
	GetTemperatureEvents := get.Events.b_CMChokeTemperatureHigh[1] 	OR
			get.Events.b_CMChokeTemperatureHigh[2]		OR
			get.Events.b_CMChokeTemperatureHigh[3]		OR
			get.Events.b_CMChokeTemperatureHigh[4] 		OR
			get.Events.b_GridChokeTemperatureHigh[1]	OR
			get.Events.b_GridChokeTemperatureHigh[2]	OR
			get.Events.b_GridChokeTemperatureHigh[3]	OR
			get.Events.b_inverterTemperatureHigh;
ELSE
	GetTemperatureEvents := get.Events.b_CMChokeTemperatureTooHigh[1] 	OR
			get.Events.b_CMChokeTemperatureTooHigh[2]	OR
			get.Events.b_CMChokeTemperatureTooHigh[3]	OR
			get.Events.b_CMChokeTemperatureTooHigh[4]	OR
			get.Events.b_GridChokeTemperatureTooHigh[1]	OR
			get.Events.b_GridChokeTemperatureTooHigh[2]	OR
			get.Events.b_GridChokeTemperatureTooHigh[3]	OR
			get.Events.b_F56TemperatureFault;
END_IF
END_METHOD

METHOD Idle : BOOL
//Inverter.controlWord.b_ChargeDC := TRUE;
//inverter.ControlWord.b_run := TRUE;

//Set powermode
inverter.powermode := ePowermodes.Droop;
inverter.r_BaseCurrentRef := 0;
inverter.r_ReactiveCurrentRef := 0;
SetVoltageFrequency(SetToIn := TRUE, VoltIN := settings.GridParams.r_GridNominalVoltage, FreqIn := settings.GridParams.r_GridNominalFrequency);
inverter.startMode := FALSE;
inverter.Island(TRUE);
Idle := get.StatusWord.b_readytooperate AND NOT get.GridcodeStatusWord.b_GridCodeTripActive;
END_METHOD

METHOD init : BOOL

VAR_INST
	
END_VAR
inverter.ControlWord.b_ChargeDC := FALSE;
inverter.ControlWord.b_run := FALSE;
inverter.ControlWord.b_Reset := TRUE;
END_METHOD

METHOD Reset : BOOL
ton_ResetPulse(IN:= NOT ton_ResetPulse.Q);
set.b_QuickstopInactive := TRUE;

Inverter.ControlWord.b_Reset := TRUE;
buscoupler.b_MCCBChargeSpring := TRUE;

IF NOT (get.events.b_GeneralFaultFlag OR get.StatusWord.b_Fault) THEN
	Inverter.ControlWord.b_Reset := FALSE;
	buscoupler.b_MCCBChargeSpring := FALSE;
END_IF

Reset := get.e_Status <> eStatusPowerModule.fault;
END_METHOD

METHOD Run : BOOL
VAR_INPUT
	Powermode			: ePowermodes;
	InverterMode		: EInvertermodes;
	InternalPowerSet		: BOOL;
END_VAR

VAR_INST
	r_DroopMin			: REAL;
	r_DroopMax			: REAL;
END_VAR
//Set powermodes
inverter.Powermode := powermode;
inverter.startMode := FALSE;


// set invertermode
CASE InverterMode OF
	eInverterModes.Afe : Inverter.AFE();
	eInverterModes.Microgrid : Inverter.Microgrid();
	eInverterModes.Island : Inverter.Island(FALSE);
END_CASE

SetVoltageFrequency(InternalPowerSet, set.r_NomVoltage, set.r_NomFrequency);

//Set absolute power and current limits of inverter
IF InternalPowerSet THEN
	inverter.r_InputActiveCurrentLimit := 100;
	inverter.r_OutputActiveCurrentLimit := 100;
	Inverter.Island(TRUE);
ELSE
	SetInverterRefs_Limits(get := get, set := set, 
		r_InputActiveCurrentLimitRef => inverter.r_InputActiveCurrentLimit,
		r_OutputActiveCurrentLimitRef => inverter.r_OutputActiveCurrentLimit,
		r_basecurrentref => inverter.r_BaseCurrentRef,
		r_ReactiveCurrentRef => inverter.r_ReactiveCurrentRef
	);
END_IF

inverter.ControlWord.b_run := TRUE;
run := get.StatusWord.b_Running;
END_METHOD

METHOD PRIVATE SetEvents
VAR_IN_OUT CONSTANT
	st_params					: ST_Powermodule_Params;
END_VAR


VAR_IN_OUT
	events						: ST_Powermodule_events;
END_VAR

VAR 
	w_Index										: WORD;
END_VAR
FOR w_Index:=1 TO 4 DO
	 LimitTrigger(
		r_IN := get.r_TemperatureCMChoke[w_Index],
		b_HighEnable:= TRUE,
		r_HighLimit:= st_Params.r_FilterTempAlarm,
		r_HighWarning:= st_params.r_FilterTempWarning,
		b_LowEnable:= FALSE,
		r_LowLimit:= 0,
		r_LowWarning:= 0,
		r_hysteresis:= 5,
		b_Warning=> get.Events.b_CMChokeTemperatureHigh[w_Index],
		b_Fault=> get.Events.b_CMChokeTemperatureTooHigh[w_Index]
		);
END_FOR

FOR w_Index:=1 TO 3 DO
	LimitTrigger(
		r_IN := get.r_TemperatureCMChoke[w_Index],
		b_HighEnable:= TRUE,
		r_HighLimit:= st_params.r_FilterTempAlarm,
		r_HighWarning:= st_params.r_FilterTempWarning,
		b_LowEnable:= FALSE,
		r_LowLimit:= 0,
		r_LowWarning:= 0,
		r_hysteresis:= 5,
		b_Warning=>get.Events.b_GridChokeTemperatureHigh[w_Index],
		b_Fault=> get.Events.b_GridChokeTemperatureTooHigh[w_Index]
	);
END_FOR

// set warning when CMS PT100 gives out of range values. 
get.Events.b_CMSTemperatureRangeWarning := NOT get.w_TemperatureFaultWord =0;

//Set fan state warning
get.Events.b_FanStateUnknownWarning := get.b_FanFb AND NOT buscoupler.b_FanOn;
get.Events.b_24VdcUVRFault := NOT get.b_MccbUvr24VdcOK AND get.b_DCcontactorFb;
END_METHOD

METHOD PRIVATE SetInverterRefs_Limits : BOOL

VAR_IN_OUT
	get 			: ST_Powermodule_get;
	set				: ST_Powermodule_set;
END_VAR

VAR_OUTPUT
	r_InputActiveCurrentLimitRef : REAL;
	r_OutputActiveCurrentLimitRef : REAL;
	r_BaseCurrentRef			: REAL;
	r_ReactiveCurrentRef		: REAL;
END_VAR

VAR_INST
	r_PLimitOverhead				: REAL := 1.1;
	fb_ActiveCurrentMeasMA			: FB_movingAverage := (length := 1000, enable := TRUE);	
	r_MaxOvercurrentFactor			: REAL;	
	r_ActivePowerRQ					: REAL;
	r_ReactivePowerRQ				: REAL;
	fb_DynamicreactiveRemainMA		: FB_movingAverage := (length := 10, enable := TRUE);
	r_reactiveMaxCurrent			: REAL;
	r_ReactiveLimitCorrection		: REAL := 1.20;
	r_NomVoltage					: REAL := 400;
	ar_Throttling					: ARRAY [1..20] OF REAL;
	fb_SmoothThrottling				: FB_CTRL_Moving_Average := (eMode := e_ctrl_mode.eCTRL_MODE_ACTIVE);
	st_params_SmoothThrottling		: ST_CTRL_MOVING_AVERAGE_PARAMS := (
		 								tCtrlCycleTime := T#1S,
										tTaskCycleTime := T#1MS,
										nSamplesToFilter := 10);
										
	 r_InputActiveCurrentLimit		: REAL;
	 r_outputActiveCurrentLimit		: REAL;
	 r_baseCurrentSetpoint			: REAL;
	 r_reactiveCurrentsetpoint		: REAL;
	 r_VoltAC						: REAL;
	 r_DynamicCurrentLimit			: REAL;
	 r_ThrottlingValueFilterTemp	: REAL;
	 r_ThrottlingValueInverterTemp	: REAL;
	 r_ThrottlingValueMindex		: REAL;
	 r_ThrottlingActual				: REAL;
	 
	 
	 ePIDctrl						: E_CTRL_Mode;
	 //Mindex limiter
	r_ActReactiveToThrottlingValue	: REAL;
	fb_PIDMindex					: FB_CTRL_PID_EXT := (emode := e_Ctrl_mode.eCTRL_MODE_ACTIVE);
	st_Params_PIDMindex				: ST_CTRL_PID_EXT_PARAMS := ( 
										tTaskCycleTime := T#1MS,
										tCtrlCycleTime := T#1MS,
										fKp	:= 0.05,
										tTn := T#500MS,
										tTd := T#0S,
										tTv := T#0MS,
										fOutMaxLimit := 0,
										fOutMinLimit := -1,
										fouterwindow := 0
										);


	//AC current limiter
	fb_RampCurrentLimit				: FB_RAMP_Dual := (Enable := TRUE, rampDown := 50, rampUp := 20);									
	fb_PIDCurrentLimit				: FB_CTRL_PID_EXT;
	st_Params_PIDCurrentLimit		: ST_CTRL_PID_EXT_PARAMS := ( 
										tTaskCycleTime := T#1MS,
										tCtrlCycleTime := T#1MS,
										fKp	:= 0.5,
										tTn := T#500MS,
										tTd := T#0MS,
										tTv := T#0MS,
										fDeadbandInput := 10
										);
										
END_VAR
IF ton_ResetPulse.Q AND NOT get.StatusWord.b_Running THEN
	ePIDctrl := e_Ctrl_mode.eCTRL_MODE_RESET;
ELSE
	ePIDctrl := e_Ctrl_mode.eCTRL_MODE_Active;	
END_IF

r_VoltAC := get.r_ACVoltageSupply;
fb_ActiveCurrentMeasMA(IN := get.r_ActiveCurrent);
r_MaxOvercurrentFactor := MIN(st_params.r_ACCurrentLimitMax / MAX(1, st_params.r_InverterRatedCurrent), set.r_overcurrentFactor);

st_params_SmoothThrottling.pWorkArray_ADR := ADR(ar_Throttling);
st_params_SmoothThrottling.nWorkArray_SIZEOF := SIZEOF(ar_Throttling);

fb_SmoothThrottling(
	fin := get.r_TemperatureMax,
	stParams := st_params_SmoothThrottling);

r_ThrottlingValueFilterTemp := scale(
		r_in:=fb_SmoothThrottling.fOut,
		 In_min:= st_params.r_FilterTempWarning,
		 In_max:= st_params.r_FilterTempAlarm,
		 Out_min:= r_MaxOvercurrentFactor,
		 Out_max:= st_params.r_ThrottlingMinimum);
		
r_ThrottlingValueInverterTemp := scale(
		r_in:=get.r_TemperatureInverter,
		 In_min:= st_params.r_InverterTempWarning,
		 In_max:= st_params.r_InverterTempAlarm,
		 Out_min:= r_MaxOvercurrentFactor,
		 Out_max:= st_params.r_ThrottlingMinimum);	

r_ThrottlingActual	:= MIN(r_ThrottlingValueInverterTemp,r_ThrottlingValueFilterTemp);	

//TOTAL AC CURRENT LIMIT
	st_Params_PIDCurrentLimit.fOutMaxLimit := st_params.r_ACCurrentLimitMax;
	st_Params_PIDCurrentLimit.fOutMinLimit := st_params.r_ACCurrentLimitMin;
	fb_RampCurrentLimit(SetToIn := NOT get.StatusWord.b_Running, IN :=  LIMIT(st_params.r_ACcurrentLimitMin, set.r_ACcurrentLimit, st_params.r_InverterRatedCurrent *  r_throttlingActual));
	fb_PIDCurrentLimit(
		eMode := ePIDctrl,
		fSetpointValue := LIMIT(fb_RampCurrentLimit.Q,get.r_ACCurrent, fb_RampCurrentLimit.Q),
		fActualValue := get.r_ACCurrent,
		stParams:= st_params_PIDCurrentLimit,
		fout => r_DynamicCurrentLimit
		);
	
	IF fb_PIDCurrentLimit.bError THEN
		r_DynamicCurrentLimit := LIMIT(st_params.r_ACcurrentLimitMin, set.r_ACcurrentLimit, st_params.r_InverterRatedCurrent *  r_throttlingActual);
	END_IF
	
	IF st_calibration.b_StartCalibration THEN
		r_DynamicCurrentLimit := 650;
	END_IF

//ACTIVE CURRENT LIMIT
	r_InputActiveCurrentLimit := LIMIT(0 , kWToCurrent(ABS(set.r_Pmin), 400), st_params.r_ACCurrentLimitMax);
	r_OutputActiveCurrentLimit := LIMIT(0 , kWToCurrent(ABS(set.r_Pmax),  400), st_params.r_ACCurrentLimitMax);

//ACTIVE SETPOINT
	r_activePowerRQ := CompensationCurve(PIN := set.r_ActivePower, QIN := get.r_ReactivePower, coef := st_calibration.PCoefficients, mode := 0);
	r_ActivePowerRQ	:= LIMIT(get.r_Pmin, r_ActivePowerRQ, get.r_Pmax);


//REACTIVE SETPOINT + MINDEX LIMIT
st_params_PIDMindex.fDeadBandInput := st_params.r_ModulationIndexLimitHyst;
	fb_PIDMindex(
		eMode := ePIDctrl,
		fsetpointvalue :=  st_params.r_ModulationIndexLimit,
		fActualValue := get.r_ModulationIndex,
		stparams := st_Params_PIDMindex
	);	
	r_ThrottlingValueMindex := fb_PIDMindex.fout + 1;
	fb_DynamicreactiveRemainMA(IN := SQRT(MAX(EXPT(r_DynamicCurrentLimit,2) - EXPT(fb_ActiveCurrentMeasMA.Q*r_ReactiveLimitCorrection ,2), 0)) * r_ThrottlingValueMindex);
	r_ReactivePowerRQ := CompensationCurve(PIN := get.r_activePower, QIN := set.r_ReactivePower, coef := st_calibration.QCoefficients, mode := 1);
	
	//to jump to PID value when throttling starts. Otherwise takes quite some time to get there.
	r_ActReactiveToThrottlingValue := kWToCurrent(r_ActivePowerRQ, get.r_ACVoltageD7) / MAX(1, fb_DynamicreactiveRemainMA.Q);
	IF get.r_ModulationIndex > MIN(100, st_params.r_ModulationIndexLimit + st_params.r_ModulationIndexLimitHyst) AND r_ThrottlingValueMindex > r_ActReactiveToThrottlingValue THEN
		fb_PIDMindex.fManSyncValue := r_ActReactiveToThrottlingValue - 1;
		fb_PIDMindex.bSync := TRUE;
	ELSE
		fb_PIDMindex.bSync := FALSE;
	END_IF
	
//power overwrites before it is converted to refs
	IF st_calibration.b_StartCalibration THEN
		r_activePowerRQ := st_calibration.r_Pset;
		r_ReactivePowerRQ	:= st_calibration.r_Qset;
	END_IF

//To currents
	r_basecurrentSetpoint := LIMIT(-r_DynamicCurrentLimit, kWToCurrent(r_ActivePowerRQ, r_VoltAC), r_DynamicCurrentLimit);
	r_reactiveCurrentSetpoint := LIMIT(-fb_DynamicreactiveRemainMA.Q, kWToCurrent(r_ReactivePowerRQ,get.r_ACVoltageD7), fb_DynamicreactiveRemainMA.Q);	

//TO REFS
	r_InputActiveCurrentLimitRef := BaseValueToRef(r_InputActiveCurrentLimit);
	r_OutputActiveCurrentLimitRef := BaseValueToRef(r_OutputActiveCurrentLimit);
	r_baseCurrentRef := BaseValueToRef(r_basecurrentSetpoint);
	r_ReactivecurrentRef:= BaseValueToRef(r_reactiveCurrentSetpoint);

get.b_LimiterActive := TRUE;
// set limter state
IF r_ThrottlingValueMindex < fb_PIDMindex.fManSyncValue THEN
	get.e_ThrottlingStatus := ePowerModuleThrottlingState.Overvoltage;
ELSIF r_ThrottlingValueFilterTemp < r_MaxOvercurrentFactor THEN
	get.e_ThrottlingStatus := ePowerModuleThrottlingState.FilterTemp;
ELSIF r_ThrottlingValueInverterTemp < r_MaxOvercurrentFactor THEN
	get.e_ThrottlingStatus := ePowerModuleThrottlingState.InverterTemp;
ELSE
	get.b_LimiterActive := FALSE;
END_IF


	
//set the final value as feedback to the get struct of the powermodule
	get.r_OverCurrentValue 	:=  r_ThrottlingActual;
	get.r_Pmin 				:= -CurrentToKw(MIN(get.r_ACcurrentLimit, r_InputActiveCurrentLimit), r_VoltAC) * r_PLimitOverhead;
	get.r_Pmax 				:= CurrentToKw(MIN(get.r_ACcurrentLimit, r_outputActiveCurrentLimit), r_VoltAC);
	get.r_ACcurrentLimit	:= MIN(set.r_ACcurrentLimit, r_DynamicCurrentLimit);
	r_reactiveMaxCurrent 	:= MIN(fb_DynamicreactiveRemainMA.Q, SQRT(MAX(EXPT(get.r_ACcurrentLimit,2) - EXPT(get.r_ActiveCurrent,2), 0)));
	get.r_Qmax				:=  CurrentToKW(r_reactiveMaxCurrent, r_VoltAC);
	get.r_Qmin				:= -get.r_Qmax;
END_METHOD

METHOD PRIVATE SetInverterSettings : BOOL

VAR_INST
	ton_GridcodeOnDelay	: TON := (PT:= T#500MS);
	ton_GridcodeOffDelay: TON := (PT:= T#0S);
	SR_GridCodeActivate	: SR; 
	
	FtrigResetDrive		: F_TRIG;
END_VAR
//set actual droop
inverter.r_BaseRefRampRate		:= set.i_PowerChangeRate;

ton_GridcodeOffDelay(IN := (get.e_InverterMode <> eInvertermodes.Afe AND NOT get.GridcodeStatusWord.b_GridCodeTripActive) OR NOT get.StatusWord.b_Running);
ton_GridcodeOnDelay(IN:= get.e_InverterMode = eInvertermodes.Afe AND set.b_gridcodeEnable AND get.StatusWord.b_ReadyToOperate);
//Set gridcodes
SR_GridCodeActivate(
	SET1 := ton_GridcodeOnDelay.Q,
	RESET := ton_GridcodeOffDelay.Q OR NOT set.b_gridcodeEnable OR NOT get.StatusWord.b_ReadyToOperate,
	);


inverter.ControlWord.b_GridCodeEnable:= SR_GridCodeActivate.Q1;
inverter.controlword.b_ExtGridcodeTrip := set.b_ExtgridCodeTrip;

//reset drive if gridcodes are set off
FtrigResetDrive(CLK:= inverter.ControlWord.b_GridCodeEnable);
IF FtrigResetDrive.Q THEN
	Reset();
END_IF

IF NOT get.StatusWord.b_Running THEN
	//Set powermode
	inverter.Island(TRUE);
	//Set voltage / frequency
	//SetVoltageFrequency(TRUE, settings.GridParams.r_GridNominalVoltage, settings.GridParams.r_GridNominalFrequency);	
END_IF
END_METHOD

METHOD PRIVATE SetParallelDrive : BOOL
IF Settings.Configuration.b_DoublePowerModule THEN
	inverter.ControlWord.b_ParallelAFE := TRUE;
ELSE
	inverter.ControlWord.b_ParallelAFE:= FALSE;
END_IF

SetParallelDrive := Settings.Configuration.b_DoublePowerModule;
END_METHOD

METHOD SetVoltageFrequency : BOOL
VAR_INPUT
	SetToIn		: BOOL;
	VoltIN		: REAL;
	FreqIN		: REAL;
END_VAR

VAR_INST
	//rTrig_SetToIN	: R_TRIG;
END_VAR

VAR_INST
	r_FrequencyDroopOffset 	: REAL;
	r_VoltageDroopOffset 	: REAL;
	//freqRamp				: FB_ramp := (b_enable := TRUE, r_rampRate := 10);
	//VoltRamp				: FB_ramp := (b_enable := TRUE, r_rampRate := 10);
END_VAR
//rTrig_SetToIN(CLK := SetToIn);
//FreqRamp(SetToIn := NOT get.StatusWord.b_Running OR rTrig_SetToIN.Q);
//VoltRamp(SetToIn := NOT get.StatusWord.b_Running OR rTrig_SetToIN.Q);
//FreqRamp.IN := FreqIN;	
//VoltRamp.IN := VoltIN;

// set gridnominal Frequency
r_FrequencyDroopOffset := FreqIN - settings.GridParams.r_GridNominalFrequency;
inverter.r_FrequencyDroopOffset := LIMIT(-2, r_FrequencyDroopOffset, 2);
// set gridnominal voltage
r_VoltageDroopOffset := VoltIN - settings.GridParams.r_GridNominalVoltage + st_params.i_VoltageOffset;
inverter.r_VoltageCorrection	:= LIMIT(-40 + st_params.i_VoltageOffset, r_VoltageDroopOffset, 40 + st_params.i_VoltageOffset);
END_METHOD

METHOD Shutdown : BOOL
VAR_INPUT
	b_Force		: BOOL := FALSE;
END_VAR

VAR_INST
	b_enableForce : BOOL := FALSE;
	currentMax : REAL;
	r_DCcurrentAbs : REAL;
	r_DCcurrent	: REAL;
END_VAR

VAR
	r_DCreleaseCurrent		: REAL := 20;
END_VAR
r_DCcurrentAbs := ABS(get.r_DCCurrent);
inverter.r_BaseCurrentRef := 0;
inverter.r_ReactiveCurrentRef := 0;

IF (b_Force OR get.StatusWord.b_Fault) THEN
	inverter.ControlWord.b_ChargeDC := FALSE;
	inverter.ControlWord.b_run := FALSE;
ELSE
	inverter.ControlWord.b_run := FALSE;
	inverter.r_OutputActiveCurrentLimit := 10;
	inverter.r_InputActiveCurrentLimit := 10;
	IF r_DCcurrentAbs < r_DCreleaseCurrent THEN
		inverter.ControlWord.b_ChargeDC := FALSE;
		buscoupler.b_MCCBChargeSpring := TRUE;	
	END_IF
END_IF

//minimum shutdown execution time.
shutdown := NOT inverter.ControlWord.b_ChargeDC AND NOT inverter.ControlWord.b_run AND NOT get.StatusWord.b_Running AND DecoupleDC();
END_METHOD

METHOD Start : BOOL

VAR_INPUT
	AFESTART : BOOL;
END_VAR

VAR_INST
	tp_RunDelay			: TP := (PT:= T#1S);
	StartupValue		:	BOOL := TRUE;
	b_RunAlready		: BOOl;
END_VAR
inverter.r_OutputActiveCurrentLimit := 520;
inverter.r_InputActiveCurrentLimit := 520; 
inverter.ControlWord.b_run := FALSE;
inverter.startMode := TRUE;

IF AFESTART THEN
	inverter.AFE();
ELSE
	inverter.Island(TRUE);
END_IF

SetVoltageFrequency(TRUE, settings.GridParams.r_GridNominalVoltage, settings.GridParams.r_GridNominalFrequency);

(*STEPS
first check if DC exists
if its yet there and checkDCvoltage gives TRUE, inverter can get to run state.
Ifnot, try precharging (if its in the system).

*)
IF get.b_MccbUvr24VdcOK THEN
	inverter.ControlWord.b_ChargeDC := get.StatusWord.b_ReadyToDCCharge;
	tp_RunDelay(in := CheckDCvoltage() AND NOT tp_RunDelay.Q);
	b_RunAlready := get.StatusWord.b_running AND get.r_ACVoltageSupply <> 0;
	inverter.ControlWord.b_run := tp_RunDelay.Q OR b_RunAlready;
END_IF


//Check if we already have DC
IF CoupleDC() THEN
	Start := get.StatusWord.b_Running;
END_IF



//OLD code, run delay and startup value might be needed -- To be tested
(*


IF CheckDCvoltage(r_BatDcVoltage) THEN
	inverter.ControlWord.b_ChargeDC := get.StatusWord.b_ReadyToDCCharge;
	inverter.ControlWord.b_run := tp_RunDelay.Q OR startupValue;
	StartupValue := FALSE;
	
	IF get.StatusWord.b_Running THEN
		tp_RunDelay(in := FALSE);
	END_IF
	Start := get.StatusWord.b_Running;
END_IF
*)
END_METHOD

END_FUNCTION_BLOCK

// ---- POUs/Objects/PowerStack/PowerModule/FB_PowerModule_Inverter.TcPOU
FUNCTION_BLOCK FB_PowerModule_Inverter
VAR_IN_OUT
	get									: ST_PowerModule_Get;
	set									: ST_Powermodule_Set;
END_VAR

VAR_IN_OUT CONSTANT
	st_params							: ST_PowerModule_params;									
END_VAR

VAR_INPUT
	b_parallelDrive						: BOOL;
	ControlWord							: ST_InverterControlWord;
	r_InputActiveCurrentLimit			: REAL;
	r_OutputActiveCurrentLimit			: REAL;
	
//current refs for power calc
	r_BaseCurrentRef					: REAL;
	r_BaseRefRampRate					: REAL;
	r_ReactiveCurrentRef				: REAL;
	r_FrequencyDroopOffset				: REAL;
	r_VoltageCorrection					: REAL;
	Powermode							: ePowermodes;
	StartMode							: BOOL;
END_VAR	

VAR
	// Local variables
	//IO variables
	a_StatusDataIN					AT %I* : ARRAY[1..2] OF UINT;
	a_ProcessDataIN					AT %I* : ARRAY[1..16] OF INT;
	a_ControlDataOUT				AT %Q* : ARRAY[1..1] OF UINT;
	a_ProcessDataOUT				AT %Q* : ARRAY[1..16] OF INT;
	
	i_InverterMode					: INT; // 0= AFE, 1= ugrid	
END_VAR

VAR_STAT
	r_DroopMax						: REAL;
	r_DroopMin						: REAL;
	r_DroopIsland					: REAL;
	
	//Power mode final
	w_StartPowerMode				: WORD;  // 0= Zero D7, 1= Zero Supply, 2= Droop, 3= iso
	w_StartVoltageMode				: WORD;	// 0= Zero D7, 1= Droop, 2= Keep reactive Ref (iso)
END_VAR


// Read data
Read();

//Watchdog Feedback and pulse
WatchdogTimer();

//Setpowermode
SetPowermode();

//Write data
Write(get, st_params);

METHOD AFE : BOOL
VAR_INPUT
END_VAR
i_invertermode	:= 0; //AFE
r_DroopMin := set.r_DroopMaximum;
r_DroopMax := set.r_DroopMaximum;
END_METHOD

METHOD PRIVATE IntPercentageToReal : REAL
VAR_INPUT
	in				: INT;
	ratedCurrent	: REAL;
END_VAR
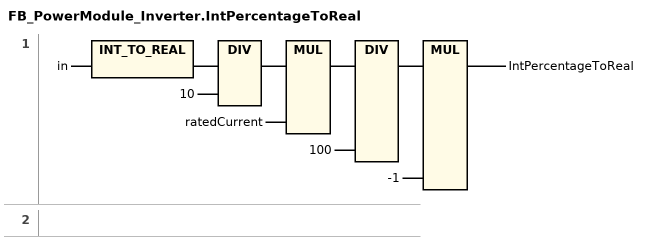
// NETWORK 1
IntPercentageToReal := (((INT_TO_REAL(in) / 10) * ratedCurrent) / 100) * -1;

// NETWORK 2
END_METHOD

METHOD Island : BOOL
VAR_INPUT
	soft	: BOOL;
END_VAR
i_invertermode := 2; //Ugrid
r_DroopMin:= set.r_DroopIslandMode;
r_DroopMax:= set.r_DroopIslandMode;


IF soft THEN
	powermode := ePowermodes.DroopZeroStart;
	r_DroopMin:= 1;
	r_DroopMax:= 1;
ELSE
	powermode := ePowermodes.Droop;
	r_DroopMin:= set.r_DroopIslandMode;
	r_DroopMax:= set.r_DroopIslandMode;
END_IF
END_METHOD

METHOD Microgrid : BOOL

VAR_INPUT
	
END_VAR
i_invertermode := 2; //Ugrid
r_DroopMin := set.r_DroopMinimum;
r_DroopMax := set.r_DroopMaximum;
END_METHOD

METHOD Read : BOOL

VAR_INST
	w_MicrogridStatusWord		: WORD;
	w_FaultStatusWord1			: WORD;
	w_FaultStatusWord2			: WORD;
	w_GridcodeStatusWord		: WORD;
	w_ModulationIndex			: WORD;
	ModulationIndexMA			: fb_MovingAverage := (enable := TRUE,  length:= 100);
END_VAR
//Convert get.RawReadData to right data type and range.
	w_MicrogridStatusWord		:= TO_WORD(a_ProcessDataIn[1]); 
	get.r_DCVoltage 			:= INT_TO_REAL(a_ProcessDataIn[2]);
	get.r_DCCurrent				:= -INT_TO_REAL(a_ProcessDataIn[3]);
	get.r_D7SyncError			:= scale(r_in:= INT_TO_REAL(a_ProcessDataIn[4]), In_min :=-3072, In_max:=3071, Out_min:=-180, Out_max:= 180);
	get.r_ActiveCurrent			:= IntPercentageToReal(a_ProcessDataIn[5], st_params.r_InverterRatedCurrent);
	get.r_ReactiveCurrent		:= IntPercentageToReal(a_ProcessDataIn[6], st_params.r_InverterRatedCurrent);
	get.r_ACVoltageD7			:= INT_TO_REAL(a_ProcessDataIn[7]);
	get.r_FrequencyD7			:= MAX(0, INT_TO_REAL(a_ProcessDataIn[8]))/100;
	get.r_TemperatureInverter	:= INT_TO_REAL(a_ProcessDataIn[9]);
	get.r_ACVoltageSupply		:= INT_TO_REAL(a_ProcessDataIn[10])/10;
	get.r_FrequencySupply		:= MAX(0, INT_TO_REAL(a_ProcessDataIn[11]))/100;
	get.r_ACCurrent				:= INT_TO_REAL(a_ProcessDataIn[12]);
	w_FaultStatusWord1			:= TO_WORD(a_ProcessDataIn[13]);
	w_FaultStatusWord2			:= TO_WORD(a_ProcessDataIn[14]);
	w_GridcodeStatusWord		:= TO_WORD(a_processDataIN[15]);
	w_modulationIndex			:= TO_WORD(a_processDataIN[16]);

ModulationIndexMA(IN := TO_REAL(w_modulationIndex)/ 10, Q => get.r_ModulationIndex);

//UNPACK General Status Word
UnpackWord(
	w_IN:= TO_WORD(a_StatusDataIn[1]),
	b0=>get.StatusWord.b_ReadyToDCCharge,
	b1=>get.StatusWord.b_ReadyToOperate,
	b2=>get.StatusWord.b_Running,
	b3=>get.StatusWord.b_Fault,
	b4=>get.StatusWord.b_RunEnabled,
	b5=>get.StatusWord.b_QuickstopNotActive,
	b6=>get.StatusWord.b_MCCBControlNotOK,
	b7=>get.StatusWord.b_Warning,
	b8=>get.StatusWord.b_DCAtReference,
	b9=>,
	b10=>get.StatusWord.b_DCAboveLimit,
	b11=>,
	b12=>,
	b13=>,
	b14=>,
	b15=>get.StatusWord.b_WatchdogFeedback,
);

get.ui_InverterCommStatus := a_StatusDataIn[2];

//UNPACK Ugridword 
UnpackWord(
	w_IN:= w_MicrogridStatusword,
	b0=>Get.UgridStatusWord.b_ChargeControlActive,
	b1=>get.UgridStatusWord.b_InternalChargingSwitchStatus,
	b2=>get.UgridStatusWord.b_MCBcontrol,
	b3=>Get.UgridStatusWord.b_MCBStatus,
	b4=>Get.UgridStatusWord.b_RunEnabled,
	b5=>Get.UgridStatusWord.b_DriveReady,
	b6=>Get.UgridStatusWord.b_AFEmodeActive,
	b7=>Get.UgridStatusWord.b_IslandModeActive,
	b8=>Get.UgridStatusWord.b_MicrogridModeActive,
	b9=>Get.UgridStatusWord.b_RunRequestActive,
	b10=>Get.UgridStatusWord.b_DriveInRunState,
	b11=>Get.UgridStatusWord.b_FaultActive,
	b12=>Get.UgridStatusWord.b_SynchronizedToD7,
	b13=>,
	b14=>Get.UgridStatusWord.b_D7MeasurementsOK,
	b15=>
);

//get mccbfb from inverter ugrid word.
Get.b_MccbFb := get.UgridStatusWord.b_MCBStatus;

//UNPACK Fault Word
UnpackWord(
	w_IN:= w_FaultStatusWord1,
	b0=>get.Events.b_F1OverCurrent,
	b1=>get.Events.b_F2OverVoltage,
	b2=>get.Events.b_F9UnderVoltage,
	b3=>get.Events.b_F91ShortCircuit,
	b4=>get.Events.b_F3EarthFault,
	b5=>,
	b6=>get.Events.b_F14UnitOverTemperature,
	b7=>get.Events.b_F56TemperatureFault,
	b8=>get.Events.b_F10LineSynchFault,
	b9=>,
	b10=>,
	b11=>get.Events.b_F52KeypadOCCommFault,
	b12=>get.Events.b_F53FieldbusFault,
	b13=>get.Events.b_F59SystembusFault,
	b14=>get.Events.b_F54SlotCommunicationFault,
	b15=>get.Events.b_F50Meas4mAFault
);

UnpackWord(
	w_IN:= w_FaultStatusWord2,
	b0=>get.Events.b_F11OutputPhaseFault,
	b1=>get.Events.b_F80ChargeFault,
	b2=>,
	b3=>,
	b4=>,
	b5=>,
	b6=>get.Events.b_F51ExternalFault,
	b7=>,
	b8=>,
	b9=>get.Events.b_F31IGBTFault,
	b10=>,
	b11=>,
	b12=>,
	b13=>,
	b14=>get.Events.b_F64MCBstateFault,
	b15=>
);

UnpackWord(
	w_IN:= w_GridcodeStatusWord,
	b0=>get.GridcodeStatusWord.b_LineVoltTripLimHigh,
	b1=>get.GridcodeStatusWord.b_LineVoltTripLimLow,
	b2=>get.GridcodeStatusWord.b_LineFreqTripLimHigh,
	b3=>get.GridcodeStatusWord.b_LineFreqTripLimLow,
	b4=>,
	b5=>,
	b6=>,
	b7=>,
	b8=>,
	b9=>,
	b10=>,
	b11=>get.GridcodeStatusWord.b_LineFreqOK,
	b12=>get.GridcodeStatusWord.b_LineVoltOK,
	b13=>get.GridcodeStatusWord.b_FRTActive,
	b14=>,
	b15=>get.GridcodeStatusWord.b_GridCodeTripActive
);


(*
INFO VACON IDs

Status word				: ID68, see ARFIF106 manual
1.Line state word		: ID3547,  (gridcode state) --> shift down
1.MicroGridSW			: ID1701, see ARFIF106 manual
2.DCVoltage				: ID1108, unit: VDC
3.DCCurrent				: ID72, Unit: Ampere DC
4.D7 Sync Error 		: ID1659, Unit: degree -3072...+3071 = -180...180 degrees.
5.ActiveCurrent			: ID1125, Unit: % of rated current
6.ReactiveCurrent 		: ID1157, Unit: % of rated current 
7.Line Voltage D7		: ID1650, Unit: VAC
8.Frequency D7			: ID1654, Unit: Hz
9.Unit temperature		: ID1109, Unit: C
10.Line voltage Supply	: ID1107, Unit: VAC
11.Frequency Supply		: ID1	, Unit: Hz
12.Total current 		: ID1104, Unit: A
13.
14.Fault Word 1		: ID1172, See ARFIF106 manual
15. 
16.

*)
END_METHOD

METHOD PRIVATE RealToInt : INT
VAR_INPUT
	in_r_Value				: REAL ;
	in_r_Res				: REAL ;
	in_i_Offset				: INT ;
END_VAR
VAR
	r_ResolutionResolved	: REAL;
	r_OffsetSolved			: REAL;
END_VAR
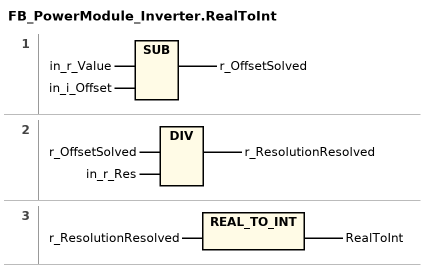
// NETWORK 1
r_OffsetSolved := in_r_Value - in_i_Offset;

// NETWORK 2
r_ResolutionResolved := r_OffsetSolved / in_r_Res;

// NETWORK 3
RealToInt := REAL_TO_INT(r_ResolutionResolved);
END_METHOD

METHOD PRIVATE SetPowerMode : BOOL
// SET Powermodes
CASE Powermode OF
	ePowermodes.DroopZeroStart : 
		get.e_PowerMode			:= ePowerModes.DroopZeroStart;
		w_StartPowerMode		:= 0;
		w_StartVoltageMode		:= 0;
	ePowermodes.Droop :
		get.e_PowerMode			:= ePowerModes.Droop;
		w_StartPowerMode		:= 2;
		w_StartVoltageMode		:= 1;
	ePowermodes.Isochronous :
		get.e_PowerMode			:= ePowerModes.Isochronous;
		w_StartPowerMode		:= 3;
		w_StartVoltageMode		:= 2;
END_CASE

IF startmode THEN
	get.e_PowerMode			:= ePowerModes.DroopZeroStart;
	w_StartPowerMode		:= 0;
	w_StartVoltageMode		:= 0;
END_IF
END_METHOD

METHOD PRIVATE UnpackWord : BOOL
VAR_INPUT
	w_IN			: WORD;
END_VAR

VAR_OUTPUT
	b0			: BOOL;
	b1			: BOOL;
	b2			: BOOL;
	b3			: BOOL;
	b4			: BOOL;
	b5			: BOOL;
	b6			: BOOL;
	b7			: BOOL;
	b8			: BOOL;
	b9			: BOOL;
	b10			: BOOL;
	b11			: BOOL;
	b12			: BOOL;
	b13			: BOOL;
	b14			: BOOL;
	b15			: BOOL;
END_VAR
b0 := w_IN.0;
b1 := w_IN.1;
b2 := w_IN.2;
b3 := w_IN.3;
b4 := w_IN.4;
b5 := w_IN.5;
b6 := w_IN.6;
b7 := w_IN.7;
b8 := w_IN.8;
b9 := w_IN.9;
b10 := w_IN.10;
b11 := w_IN.11;
b12 := w_IN.12;
b13 := w_IN.13;
b14 := w_IN.14;
b15 := w_IN.15;
END_METHOD

METHOD PRIVATE WatchdogTimer : BOOL 

VAR_INST
	t_WatchdogFb1				: TON;
	t_WatchdogFB2				: TON;
	t_WatchdogTimer1			: TON;
	t_WatchdogTimer2			: TON;
	b_WatchdogPulseFalse		: BOOL;
END_VAR
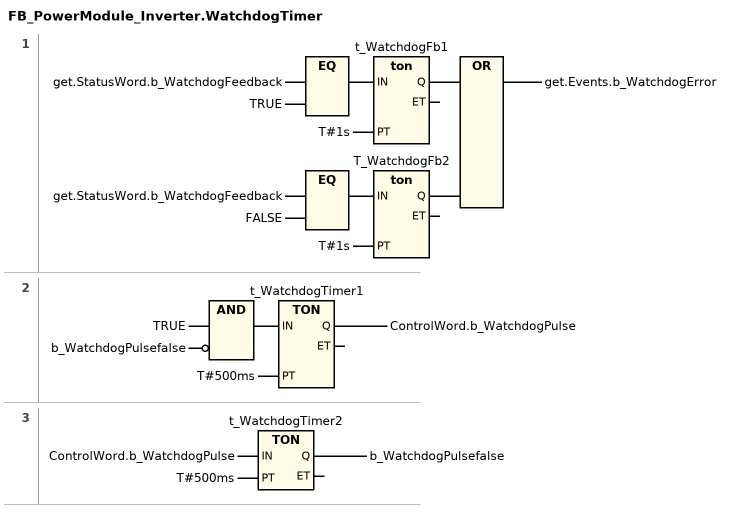
// NETWORK 1
t_WatchdogFb1(IN := get.StatusWord.b_WatchdogFeedback = TRUE, PT := T#1s); // ton
T_WatchdogFb2(IN := get.StatusWord.b_WatchdogFeedback = FALSE, PT := T#1s); // ton
get.Events.b_WatchdogError := t_WatchdogFb1.Q OR T_WatchdogFb2.Q;

// NETWORK 2
t_WatchdogTimer1(IN := TRUE AND NOT b_WatchdogPulsefalse, PT := T#500ms); // TON
ControlWord.b_WatchdogPulse := t_WatchdogTimer1.Q;

// NETWORK 3
t_WatchdogTimer2(IN := ControlWord.b_WatchdogPulse, PT := T#500ms); // TON
b_WatchdogPulsefalse := t_WatchdogTimer2.Q;
END_METHOD

METHOD Write : BOOL
VAR_IN_OUT
	get : ST_Powermodule_get;
END_VAR

VAR_IN_OUT CONSTANT
	st_params							: ST_PowerModule_params;									
END_VAR

VAR_INST
	b_rampEnable						: BOOL := TRUE;		
	fb_Ramp_OutactLim					: FB_Ramp := (r_RampRate:=100);
	fb_Ramp_InActLim					: FB_Ramp := (r_RampRate:=100);	
	
	r_FreqDroopAct						: REAL;
	r_VoltDroopAct						: REAL;
END_VAR
fb_Ramp_OutActLim(IN:=r_OutputActiveCurrentLimit, b_enable:= b_rampEnable);
fb_Ramp_InActLim(IN:=r_InputActiveCurrentLimit, b_enable:= b_rampEnable);

IF get.e_PowerMode = ePowerModes.Isochronous OR startmode THEN
	r_FreqDroopAct := set.r_DroopMaximum;
	r_VoltDroopAct := set.r_DroopMaximum;
ELSE
	r_FreqDroopAct := LIMIT(r_DroopMin, set.r_FrequencyDroop, r_DroopMax);
	r_VoltDroopAct := LIMIT(r_DroopMin, set.r_VoltageDroop, r_DroopMax);
END_IF


//get
get.controldata.Controlword := controlword;
get.controldata.i_invertermode := i_invertermode;
get.controldata.i_BaseCurrentRef := RealToInt(r_BaseCurrentRef, 0.1, 0);
get.controldata.i_ReactiveCurrentRef:= RealToInt(-r_ReactiveCurrentRef, 0.1, 0);
get.controldata.i_FrequencyDroop := RealToInt(r_FreqDroopAct , 0.002, 0); // Convert percentage to  mHz and rescale. So +100% ==> +5000.0 mHz
get.controldata.i_VoltageDroop := RealToInt(r_VoltDroopAct, 0.01, 0);
get.controldata.i_FrequencyDroopOffset := RealToInt(r_FrequencyDroopOffset, 0.01, 0);
get.controldata.i_VoltageCorrection := RealToInt(r_VoltageCorrection, 1, 0);
get.controldata.i_BaseRefRampRate := LIMIT(-1, RealToInt(r_BaseRefRampRate, 1, 0),10000);
get.controldata.i_StartPowerMode := WORD_TO_INT(w_StartPowerMode);
get.controldata.i_StartVoltageMode := WORD_TO_INT(w_StartVoltageMode);
get.controldata.i_OutActCurrentLimit := RealToInt(fb_Ramp_OutActLim.Q, 0.1, 0);
get.controldata.i_InActCurrentLimit := RealToInt(fb_Ramp_InActLim.Q, 0.1, 0);
get.controldata.i_DCVramprate :=  LIMIT(-1, st_params.i_DCVramprate, 10000);
get.r_FrequencyDroop := r_FreqDroopAct;
get.r_VoltageDroop := r_VoltDroopAct;



get.controldata.ui_controlwordvalue	:= PackWord(
	b0:=ControlWord.b_ChargeDC,
	b1:= TRUE, //b_MccbCloseEnable,
	b2:= TRUE,//set.b_QuickstopInactive,
	b3:= ControlWord.b_Run,
	b4:=TRUE, //b_OutputpowerLimits,
	b5:=TRUE, //b_PowerIncreaseEnable,
	b6:=TRUE,//b_InputpowerLimits,
	b7:= ControlWord.b_Reset,
	b8:=0,
	b9:=0,
	b10:= ControlWord.b_FieldbusControlEnable,
	b11:= ControlWord.b_WatchdogPulse,
	b12:= ControlWord.b_ParallelAFE, // ID1501
	b13:= ControlWord.b_GridCodeEnable,
	b14:= ControlWord.b_ExtGridcodeTrip, // ID3310
	b15:=0
);

